  MoveL 1251 to (509.44, 499.54, 1.8) mm, rotated rx 0 ry 90 rz 0 deg; joints [-11.786, -26.31, 109.715, -15.811, -82.79, 51.021]
  Set speed (120.0 mm/s)
  MoveL 1252 to (509.32, 490.68, 1.8) mm, rotated rx 0 ry 90 rz 0 deg; joints [-10.985, -26.346, 109.945, -14.998, -82.953, 50.882]
  Set speed (30.0 mm/s)
  Call Extruder(0.767)
  MoveL 1253 to (490.68, 509.32, 1.8) mm, rotated rx 0 ry 90 rz 0 deg; joints [-13.056, -26.6, 111.69, -17.036, -84.442, 50.665]
  MoveL 1254 to (490.56, 509.44, 1.8) mm, rotated rx 0 ry 90 rz 0 deg; joints [-13.07, -26.602, 111.701, -17.049, -84.451, 50.664]
  Set speed (120.0 mm/s)
  MoveL 1255 to (490.4, 509.6, 1.8) mm, rotated rx 0 ry 90 rz 0 deg; joints [-13.088, -26.604, 111.715, -17.067, -84.463, 50.661]
  Set speed (15.0 mm/s)
  Call Extruder(0.559)
  MoveL 1256 to (490.4, 490.4, 1.8) mm, rotated rx 0 ry 90 rz 0 deg; joints [-11.303, -26.669, 112.203, -15.264, -84.829, 50.403]
  MoveL 1257 to (509.6, 490.4, 1.8) mm, rotated rx 0 ry 90 rz 0 deg; joints [-10.955, -26.341, 109.917, -14.969, -82.93, 50.884]
  MoveL 1258 to (509.6, 509.6, 1.8) mm, rotated rx 0 ry 90 rz 0 deg; joints [-12.688, -26.265, 109.434, -16.729, -82.593, 51.19]
  MoveL 1259 to (490.4, 509.6, 1.8) mm, rotated rx 0 ry 90 rz 0 deg; joints [-13.088, -26.604, 111.715, -17.067, -84.463, 50.661]
  Set speed (120.0 mm/s)
  MoveL 1260 to (490.4, 509.2, 1.8) mm, rotated rx 0 ry 90 rz 0 deg; joints [-13.051, -26.605, 111.726, -17.03, -84.471, 50.656]
  Set speed (1000.0 mm/s)
  MoveL 1261 to (491.1, 508.9, 1.8) mm, rotated rx 0 ry 90 rz 0 deg; joints [-13.008, -26.595, 111.652, -16.989, -84.409, 50.671]
  Set speed (1000.0 mm/s)
  MoveL 1262 to (490.68, 490.68, 1.8) mm, rotated rx 0 ry 90 rz 0 deg; joints [-11.324, -26.664, 112.164, -15.286, -84.797, 50.413]
  Set speed (1000.0 mm/s)
  MoveL 1263 to (490.68, 490.68, 1.9) mm, rotated rx 0 ry 90 rz 0 deg; joints [-11.324, -26.674, 112.169, -15.286, -84.792, 50.415]
  Set speed (30.0 mm/s)
  Call Extruder(0.767)
  MoveL 1264 to (509.32, 509.32, 1.9) mm, rotated rx 0 ry 90 rz 0 deg; joints [-12.669, -26.282, 109.481, -16.708, -82.621, 51.179]
  MoveL 1265 to (509.44, 509.44, 1.9) mm, rotated rx 0 ry 90 rz 0 deg; joints [-12.677, -26.279, 109.463, -16.717, -82.606, 51.185]
  Set speed (120.0 mm/s)
  MoveL 1266 to (509.32, 500.58, 1.9) mm, rotated rx 0 ry 90 rz 0 deg; joints [-11.882, -26.319, 109.709, -15.909, -82.779, 51.036]
  Set speed (30.0 mm/s)
  Call Extruder(0.360)
  MoveL 1267 to (500.58, 509.32, 1.9) mm, rotated rx 0 ry 90 rz 0 deg; joints [-12.847, -26.444, 110.525, -16.857, -83.471, 50.942]
  Set speed (120.0 mm/s)
  MoveL 1268 to (499.42, 509.32, 1.9) mm, rotated rx 0 ry 90 rz 0 deg; joints [-12.872, -26.464, 110.663, -16.877, -83.584, 50.91]
  Set speed (30.0 mm/s)
  Call Extruder(0.360)
  MoveL 1269 to (490.68, 500.58, 1.9) mm, rotated rx 0 ry 90 rz 0 deg; joints [-12.247, -26.642, 111.926, -16.218, -84.609, 50.544]
  Set speed (120.0 mm/s)
  MoveL 1270 to (490.68, 499.42, 1.9) mm, rotated rx 0 ry 90 rz 0 deg; joints [-12.139, -26.646, 111.955, -16.109, -84.631, 50.528]
  Set speed (30.0 mm/s)
  MoveL 1271 to (499.42, 490.68, 1.9) mm, rotated rx 0 ry 90 rz 0 deg; joints [-11.163, -26.533, 111.134, -15.147, -83.926, 50.637]
  Set speed (120.0 mm/s)
  MoveL 1272 to (500.58, 490.68, 1.9) mm, rotated rx 0 ry 90 rz 0 deg; joints [-11.141, -26.513, 110.996, -15.129, -83.811, 50.666]
  Set speed (30.0 mm/s)
  Call Extruder(0.360)
  MoveL 1273 to (509.32, 499.42, 1.9) mm, rotated rx 0 ry 90 rz 0 deg; joints [-11.777, -26.323, 109.738, -15.802, -82.8, 51.018]
  MoveL 1274 to (509.44, 499.54, 1.9) mm, rotated rx 0 ry 90 rz 0 deg; joints [-11.786, -26.32, 109.721, -15.812, -82.785, 51.023]
  Set speed (120.0 mm/s)
  MoveL 1275 to (509.32, 490.68, 1.9) mm, rotated rx 0 ry 90 rz 0 deg; joints [-10.985, -26.356, 109.95, -14.999, -82.948, 50.883]
  Set speed (30.0 mm/s)
  Call Extruder(0.767)
  MoveL 1276 to (490.68, 509.32, 1.9) mm, rotated rx 0 ry 90 rz 0 deg; joints [-13.056, -26.611, 111.695, -17.036, -84.437, 50.667]
  MoveL 1277 to (490.56, 509.44, 1.9) mm, rotated rx 0 ry 90 rz 0 deg; joints [-13.07, -26.612, 111.706, -17.049, -84.446, 50.665]
  Set speed (120.0 mm/s)
  MoveL 1278 to (490.4, 509.6, 1.9) mm, rotated rx 0 ry 90 rz 0 deg; joints [-13.088, -26.614, 111.72, -17.067, -84.458, 50.663]
  Set speed (15.0 mm/s)
  Call Extruder(0.559)
  MoveL 1279 to (490.4, 490.4, 1.9) mm, rotated rx 0 ry 90 rz 0 deg; joints [-11.303, -26.679, 112.209, -15.264, -84.824, 50.404]
  MoveL 1280 to (509.6, 490.4, 1.9) mm, rotated rx 0 ry 90 rz 0 deg; joints [-10.955, -26.352, 109.923, -14.969, -82.925, 50.886]
  MoveL 1281 to (509.6, 509.6, 1.9) mm, rotated rx 0 ry 90 rz 0 deg; joints [-12.688, -26.276, 109.44, -16.729, -82.588, 51.192]
  MoveL 1282 to (490.4, 509.6, 1.9) mm, rotated rx 0 ry 90 rz 0 deg; joints [-13.088, -26.614, 111.72, -17.067, -84.458, 50.663]
  Set speed (120.0 mm/s)
  MoveL 1283 to (490.4, 509.2, 1.9) mm, rotated rx 0 ry 90 rz 0 deg; joints [-13.051, -26.616, 111.731, -17.03, -84.466, 50.657]
  Set speed (1000.0 mm/s)
  MoveL 1284 to (491.1, 508.9, 1.9) mm, rotated rx 0 ry 90 rz 0 deg; joints [-13.008, -26.606, 111.657, -16.989, -84.404, 50.672]
  Set speed (1000.0 mm/s)
  MoveL 1285 to (490.68, 490.68, 1.9) mm, rotated rx 0 ry 90 rz 0 deg; joints [-11.324, -26.674, 112.169, -15.286, -84.792, 50.415]
  Set speed (1000.0 mm/s)
  MoveL 1286 to (490.68, 490.68, 2) mm, rotated rx 0 ry 90 rz 0 deg; joints [-11.324, -26.685, 112.175, -15.286, -84.786, 50.416]
  Set speed (30.0 mm/s)
  Call Extruder(0.767)
  MoveL 1287 to (509.32, 509.32, 2) mm, rotated rx 0 ry 90 rz 0 deg; joints [-12.669, -26.293, 109.486, -16.708, -82.616, 51.181]
  MoveL 1288 to (509.44, 509.44, 2) mm, rotated rx 0 ry 90 rz 0 deg; joints [-12.677, -26.29, 109.468, -16.718, -82.602, 51.186]
  Set speed (120.0 mm/s)
  MoveL 1289 to (509.32, 500.58, 2) mm, rotated rx 0 ry 90 rz 0 deg; joints [-11.882, -26.329, 109.715, -15.909, -82.774, 51.038]
  Set speed (30.0 mm/s)
  Call Extruder(0.360)
  MoveL 1290 to (500.58, 509.32, 2) mm, rotated rx 0 ry 90 rz 0 deg; joints [-12.847, -26.454, 110.53, -16.857, -83.466, 50.943]
  Set speed (120.0 mm/s)
  MoveL 1291 to (499.42, 509.32, 2) mm, rotated rx 0 ry 90 rz 0 deg; joints [-12.872, -26.475, 110.668, -16.878, -83.579, 50.911]
  Set speed (30.0 mm/s)
  Call Extruder(0.360)
  MoveL 1292 to (490.68, 500.58, 2) mm, rotated rx 0 ry 90 rz 0 deg; joints [-12.247, -26.653, 111.931, -16.218, -84.603, 50.545]
  Set speed (120.0 mm/s)
  MoveL 1293 to (490.68, 499.42, 2) mm, rotated rx 0 ry 90 rz 0 deg; joints [-12.139, -26.657, 111.961, -16.109, -84.626, 50.53]
  Set speed (30.0 mm/s)
  MoveL 1294 to (499.42, 490.68, 2) mm, rotated rx 0 ry 90 rz 0 deg; joints [-11.163, -26.543, 111.14, -15.147, -83.921, 50.638]
  Set speed (120.0 mm/s)
  MoveL 1295 to (500.58, 490.68, 2) mm, rotated rx 0 ry 90 rz 0 deg; joints [-11.141, -26.523, 111.002, -15.129, -83.806, 50.667]
  Set speed (30.0 mm/s)
  Call Extruder(0.360)
  MoveL 1296 to (509.32, 499.42, 2) mm, rotated rx 0 ry 90 rz 0 deg; joints [-11.777, -26.334, 109.744, -15.802, -82.795, 51.019]
  MoveL 1297 to (509.44, 499.54, 2) mm, rotated rx 0 ry 90 rz 0 deg; joints [-11.786, -26.331, 109.726, -15.812, -82.781, 51.024]
  Set speed (120.0 mm/s)
  MoveL 1298 to (509.32, 490.68, 2) mm, rotated rx 0 ry 90 rz 0 deg; joints [-10.985, -26.367, 109.955, -14.999, -82.943, 50.884]
  Set speed (30.0 mm/s)
  Call Extruder(0.767)
  MoveL 1299 to (490.68, 509.32, 2) mm, rotated rx 0 ry 90 rz 0 deg; joints [-13.056, -26.621, 111.7, -17.036, -84.432, 50.668]
  MoveL 1300 to (490.56, 509.44, 2) mm, rotated rx 0 ry 90 rz 0 deg; joints [-13.07, -26.623, 111.712, -17.05, -84.441, 50.667]
  Set speed (120.0 mm/s)
  MoveL 1301 to (490.4, 509.6, 2) mm, rotated rx 0 ry 90 rz 0 deg; joints [-13.088, -26.625, 111.726, -17.067, -84.453, 50.664]
  Set speed (15.0 mm/s)
  Call Extruder(0.559)
  MoveL 1302 to (490.4, 490.4, 2) mm, rotated rx 0 ry 90 rz 0 deg; joints [-11.303, -26.69, 112.214, -15.264, -84.819, 50.405]
  MoveL 1303 to (509.6, 490.4, 2) mm, rotated rx 0 ry 90 rz 0 deg; joints [-10.955, -26.362, 109.928, -14.969, -82.92, 50.887]
  MoveL 1304 to (509.6, 509.6, 2) mm, rotated rx 0 ry 90 rz 0 deg; joints [-12.688, -26.286, 109.445, -16.729, -82.583, 51.193]
  MoveL 1305 to (490.4, 509.6, 2) mm, rotated rx 0 ry 90 rz 0 deg; joints [-13.088, -26.625, 111.726, -17.067, -84.453, 50.664]
  Set speed (120.0 mm/s)
  MoveL 1306 to (490.4, 509.2, 2) mm, rotated rx 0 ry 90 rz 0 deg; joints [-13.051, -26.626, 111.737, -17.03, -84.461, 50.659]
  Set speed (1000.0 mm/s)
  MoveL 1307 to (491.1, 508.9, 2) mm, rotated rx 0 ry 90 rz 0 deg; joints [-13.008, -26.616, 111.662, -16.989, -84.399, 50.674]
  Set speed (1000.0 mm/s)
  MoveL 1308 to (490.68, 490.68, 2) mm, rotated rx 0 ry 90 rz 0 deg; joints [-11.324, -26.685, 112.175, -15.286, -84.786, 50.416]
  Set speed (1000.0 mm/s)
  MoveL 1309 to (490.68, 490.68, 2.1) mm, rotated rx 0 ry 90 rz 0 deg; joints [-11.324, -26.695, 112.18, -15.286, -84.781, 50.417]
  Set speed (30.0 mm/s)
  Call Extruder(0.767)
  MoveL 1310 to (509.32, 509.32, 2.1) mm, rotated rx 0 ry 90 rz 0 deg; joints [-12.669, -26.303, 109.491, -16.709, -82.611, 51.182]
  MoveL 1311 to (509.44, 509.44, 2.1) mm, rotated rx 0 ry 90 rz 0 deg; joints [-12.677, -26.3, 109.473, -16.718, -82.597, 51.188]
  Set speed (120.0 mm/s)
  MoveL 1312 to (509.32, 500.58, 2.1) mm, rotated rx 0 ry 90 rz 0 deg; joints [-11.882, -26.339, 109.72, -15.909, -82.769, 51.039]
  Set speed (30.0 mm/s)
  Call Extruder(0.360)
  MoveL 1313 to (500.58, 509.32, 2.1) mm, rotated rx 0 ry 90 rz 0 deg; joints [-12.847, -26.465, 110.536, -16.857, -83.462, 50.945]
  Set speed (120.0 mm/s)
  MoveL 1314 to (499.42, 509.32, 2.1) mm, rotated rx 0 ry 90 rz 0 deg; joints [-12.872, -26.485, 110.673, -16.878, -83.574, 50.913]
  Set speed (30.0 mm/s)
  Call Extruder(0.360)
  MoveL 1315 to (490.68, 500.58, 2.1) mm, rotated rx 0 ry 90 rz 0 deg; joints [-12.247, -26.663, 111.937, -16.218, -84.598, 50.547]
  Set speed (120.0 mm/s)
  MoveL 1316 to (490.68, 499.42, 2.1) mm, rotated rx 0 ry 90 rz 0 deg; joints [-12.139, -26.667, 111.966, -16.109, -84.621, 50.531]
  Set speed (30.0 mm/s)
  MoveL 1317 to (499.42, 490.68, 2.1) mm, rotated rx 0 ry 90 rz 0 deg; joints [-11.163, -26.554, 111.145, -15.147, -83.916, 50.64]
  Set speed (120.0 mm/s)
  MoveL 1318 to (500.58, 490.68, 2.1) mm, rotated rx 0 ry 90 rz 0 deg; joints [-11.141, -26.534, 111.007, -15.129, -83.801, 50.669]
  Set speed (30.0 mm/s)
  Call Extruder(0.360)
  MoveL 1319 to (509.32, 499.42, 2.1) mm, rotated rx 0 ry 90 rz 0 deg; joints [-11.777, -26.344, 109.749, -15.803, -82.79, 51.02]
  MoveL 1320 to (509.44, 499.54, 2.1) mm, rotated rx 0 ry 90 rz 0 deg; joints [-11.786, -26.341, 109.731, -15.812, -82.776, 51.026]
  Set speed (120.0 mm/s)
  MoveL 1321 to (509.32, 490.68, 2.1) mm, rotated rx 0 ry 90 rz 0 deg; joints [-10.985, -26.377, 109.961, -14.999, -82.938, 50.886]
  Set speed (30.0 mm/s)
  Call Extruder(0.767)
  MoveL 1322 to (490.68, 509.32, 2.1) mm, rotated rx 0 ry 90 rz 0 deg; joints [-13.056, -26.632, 111.706, -17.036, -84.427, 50.67]
  MoveL 1323 to (490.56, 509.44, 2.1) mm, rotated rx 0 ry 90 rz 0 deg; joints [-13.07, -26.634, 111.717, -17.05, -84.436, 50.668]
  Set speed (120.0 mm/s)
  MoveL 1324 to (490.4, 509.6, 2.1) mm, rotated rx 0 ry 90 rz 0 deg; joints [-13.088, -26.636, 111.731, -17.067, -84.448, 50.666]
  Set speed (15.0 mm/s)
  Call Extruder(0.559)
  MoveL 1325 to (490.4, 490.4, 2.1) mm, rotated rx 0 ry 90 rz 0 deg; joints [-11.303, -26.701, 112.219, -15.264, -84.814, 50.407]
  MoveL 1326 to (509.6, 490.4, 2.1) mm, rotated rx 0 ry 90 rz 0 deg; joints [-10.955, -26.373, 109.933, -14.969, -82.915, 50.888]
  MoveL 1327 to (509.6, 509.6, 2.1) mm, rotated rx 0 ry 90 rz 0 deg; joints [-12.688, -26.296, 109.45, -16.729, -82.578, 51.195]
  MoveL 1328 to (490.4, 509.6, 2.1) mm, rotated rx 0 ry 90 rz 0 deg; joints [-13.088, -26.636, 111.731, -17.067, -84.448, 50.666]
  Set speed (120.0 mm/s)
  MoveL 1329 to (490.4, 509.2, 2.1) mm, rotated rx 0 ry 90 rz 0 deg; joints [-13.051, -26.637, 111.742, -17.03, -84.456, 50.66]
  Set speed (1000.0 mm/s)
  MoveL 1330 to (491.1, 508.9, 2.1) mm, rotated rx 0 ry 90 rz 0 deg; joints [-13.008, -26.627, 111.668, -16.989, -84.394, 50.676]
  Set speed (1000.0 mm/s)
  MoveL 1331 to (490.68, 490.68, 2.1) mm, rotated rx 0 ry 90 rz 0 deg; joints [-11.324, -26.695, 112.18, -15.286, -84.781, 50.417]
  Set speed (1000.0 mm/s)
  MoveL 1332 to (490.68, 490.68, 2.2) mm, rotated rx 0 ry 90 rz 0 deg; joints [-11.324, -26.706, 112.185, -15.286, -84.776, 50.419]
  Set speed (30.0 mm/s)
  Call Extruder(0.767)
  MoveL 1333 to (509.32, 509.32, 2.2) mm, rotated rx 0 ry 90 rz 0 deg; joints [-12.669, -26.314, 109.497, -16.709, -82.606, 51.184]
  MoveL 1334 to (509.44, 509.44, 2.2) mm, rotated rx 0 ry 90 rz 0 deg; joints [-12.677, -26.311, 109.479, -16.718, -82.592, 51.189]
  Set speed (120.0 mm/s)
  MoveL 1335 to (509.32, 500.58, 2.2) mm, rotated rx 0 ry 90 rz 0 deg; joints [-11.882, -26.35, 109.725, -15.909, -82.765, 51.04]
  Set speed (30.0 mm/s)
  Call Extruder(0.360)
  MoveL 1336 to (500.58, 509.32, 2.2) mm, rotated rx 0 ry 90 rz 0 deg; joints [-12.847, -26.475, 110.541, -16.858, -83.457, 50.946]
  Set speed (120.0 mm/s)
  MoveL 1337 to (499.42, 509.32, 2.2) mm, rotated rx 0 ry 90 rz 0 deg; joints [-12.872, -26.496, 110.679, -16.878, -83.569, 50.914]
  Set speed (30.0 mm/s)
  Call Extruder(0.360)
  MoveL 1338 to (490.68, 500.58, 2.2) mm, rotated rx 0 ry 90 rz 0 deg; joints [-12.247, -26.674, 111.942, -16.218, -84.593, 50.548]
  Set speed (120.0 mm/s)
  MoveL 1339 to (490.68, 499.42, 2.2) mm, rotated rx 0 ry 90 rz 0 deg; joints [-12.139, -26.678, 111.972, -16.109, -84.616, 50.533]
  Set speed (30.0 mm/s)
  MoveL 1340 to (499.42, 490.68, 2.2) mm, rotated rx 0 ry 90 rz 0 deg; joints [-11.163, -26.564, 111.15, -15.147, -83.911, 50.641]
  Set speed (120.0 mm/s)
  MoveL 1341 to (500.58, 490.68, 2.2) mm, rotated rx 0 ry 90 rz 0 deg; joints [-11.141, -26.545, 111.012, -15.129, -83.796, 50.67]
  Set speed (30.0 mm/s)
  Call Extruder(0.360)
  MoveL 1342 to (509.32, 499.42, 2.2) mm, rotated rx 0 ry 90 rz 0 deg; joints [-11.777, -26.355, 109.754, -15.803, -82.785, 51.022]
  MoveL 1343 to (509.44, 499.54, 2.2) mm, rotated rx 0 ry 90 rz 0 deg; joints [-11.786, -26.352, 109.737, -15.812, -82.771, 51.027]
  Set speed (120.0 mm/s)
  MoveL 1344 to (509.32, 490.68, 2.2) mm, rotated rx 0 ry 90 rz 0 deg; joints [-10.985, -26.388, 109.966, -14.999, -82.933, 50.887]
  Set speed (30.0 mm/s)
  Call Extruder(0.767)
  MoveL 1345 to (490.68, 509.32, 2.2) mm, rotated rx 0 ry 90 rz 0 deg; joints [-13.056, -26.643, 111.711, -17.036, -84.422, 50.671]
  MoveL 1346 to (490.56, 509.44, 2.2) mm, rotated rx 0 ry 90 rz 0 deg; joints [-13.07, -26.644, 111.722, -17.05, -84.431, 50.67]
  Set speed (120.0 mm/s)
  MoveL 1347 to (490.4, 509.6, 2.2) mm, rotated rx 0 ry 90 rz 0 deg; joints [-13.088, -26.646, 111.736, -17.068, -84.443, 50.668]
  Set speed (15.0 mm/s)
  Call Extruder(0.559)
  MoveL 1348 to (490.4, 490.4, 2.2) mm, rotated rx 0 ry 90 rz 0 deg; joints [-11.303, -26.711, 112.225, -15.264, -84.809, 50.408]
  MoveL 1349 to (509.6, 490.4, 2.2) mm, rotated rx 0 ry 90 rz 0 deg; joints [-10.955, -26.383, 109.939, -14.969, -82.91, 50.89]
  MoveL 1350 to (509.6, 509.6, 2.2) mm, rotated rx 0 ry 90 rz 0 deg; joints [-12.688, -26.307, 109.456, -16.73, -82.574, 51.196]
  MoveL 1351 to (490.4, 509.6, 2.2) mm, rotated rx 0 ry 90 rz 0 deg; joints [-13.088, -26.646, 111.736, -17.068, -84.443, 50.668]
  Set speed (120.0 mm/s)
  MoveL 1352 to (490.4, 509.2, 2.2) mm, rotated rx 0 ry 90 rz 0 deg; joints [-13.051, -26.648, 111.747, -17.03, -84.451, 50.662]
  Set speed (1000.0 mm/s)
  MoveL 1353 to (491.1, 508.9, 2.2) mm, rotated rx 0 ry 90 rz 0 deg; joints [-13.008, -26.637, 111.673, -16.989, -84.389, 50.677]
  Set speed (1000.0 mm/s)
  MoveL 1354 to (490.68, 490.68, 2.2) mm, rotated rx 0 ry 90 rz 0 deg; joints [-11.324, -26.706, 112.185, -15.286, -84.776, 50.419]
  Set speed (1000.0 mm/s)
  MoveL 1355 to (490.68, 490.68, 2.3) mm, rotated rx 0 ry 90 rz 0 deg; joints [-11.324, -26.717, 112.191, -15.286, -84.771, 50.42]
  Set speed (30.0 mm/s)
  Call Extruder(0.767)
  MoveL 1356 to (509.32, 509.32, 2.3) mm, rotated rx 0 ry 90 rz 0 deg; joints [-12.669, -26.324, 109.502, -16.709, -82.601, 51.185]
  MoveL 1357 to (509.44, 509.44, 2.3) mm, rotated rx 0 ry 90 rz 0 deg; joints [-12.677, -26.321, 109.484, -16.718, -82.587, 51.191]
  Set speed (120.0 mm/s)
  MoveL 1358 to (509.32, 500.58, 2.3) mm, rotated rx 0 ry 90 rz 0 deg; joints [-11.882, -26.36, 109.731, -15.909, -82.76, 51.042]
  Set speed (30.0 mm/s)
  Call Extruder(0.360)
  MoveL 1359 to (500.58, 509.32, 2.3) mm, rotated rx 0 ry 90 rz 0 deg; joints [-12.847, -26.486, 110.546, -16.858, -83.452, 50.948]
  Set speed (120.0 mm/s)
  MoveL 1360 to (499.42, 509.32, 2.3) mm, rotated rx 0 ry 90 rz 0 deg; joints [-12.872, -26.506, 110.684, -16.878, -83.565, 50.916]
  Set speed (30.0 mm/s)
  Call Extruder(0.360)
  MoveL 1361 to (490.68, 500.58, 2.3) mm, rotated rx 0 ry 90 rz 0 deg; joints [-12.247, -26.685, 111.947, -16.218, -84.588, 50.55]
  Set speed (120.0 mm/s)
  MoveL 1362 to (490.68, 499.42, 2.3) mm, rotated rx 0 ry 90 rz 0 deg; joints [-12.139, -26.688, 111.977, -16.109, -84.61, 50.534]
  Set speed (30.0 mm/s)
  MoveL 1363 to (499.42, 490.68, 2.3) mm, rotated rx 0 ry 90 rz 0 deg; joints [-11.163, -26.575, 111.156, -15.147, -83.906, 50.642]
  Set speed (120.0 mm/s)
  MoveL 1364 to (500.58, 490.68, 2.3) mm, rotated rx 0 ry 90 rz 0 deg; joints [-11.141, -26.555, 111.018, -15.13, -83.791, 50.671]
  Set speed (30.0 mm/s)
  Call Extruder(0.360)
  MoveL 1365 to (509.32, 499.42, 2.3) mm, rotated rx 0 ry 90 rz 0 deg; joints [-11.777, -26.365, 109.76, -15.803, -82.78, 51.023]
  MoveL 1366 to (509.44, 499.54, 2.3) mm, rotated rx 0 ry 90 rz 0 deg; joints [-11.786, -26.362, 109.742, -15.812, -82.766, 51.028]
  Set speed (120.0 mm/s)
  MoveL 1367 to (509.32, 490.68, 2.3) mm, rotated rx 0 ry 90 rz 0 deg; joints [-10.985, -26.398, 109.971, -14.999, -82.928, 50.888]
  Set speed (30.0 mm/s)
  Call Extruder(0.767)
  MoveL 1368 to (490.68, 509.32, 2.3) mm, rotated rx 0 ry 90 rz 0 deg; joints [-13.056, -26.653, 111.717, -17.036, -84.417, 50.673]
  MoveL 1369 to (490.56, 509.44, 2.3) mm, rotated rx 0 ry 90 rz 0 deg; joints [-13.07, -26.655, 111.728, -17.05, -84.426, 50.671]
  Set speed (120.0 mm/s)
  MoveL 1370 to (490.4, 509.6, 2.3) mm, rotated rx 0 ry 90 rz 0 deg; joints [-13.088, -26.657, 111.742, -17.068, -84.438, 50.669]
  Set speed (15.0 mm/s)
  Call Extruder(0.559)
  MoveL 1371 to (490.4, 490.4, 2.3) mm, rotated rx 0 ry 90 rz 0 deg; joints [-11.303, -26.722, 112.23, -15.265, -84.804, 50.41]
  MoveL 1372 to (509.6, 490.4, 2.3) mm, rotated rx 0 ry 90 rz 0 deg; joints [-10.955, -26.394, 109.944, -14.969, -82.905, 50.891]
  MoveL 1373 to (509.6, 509.6, 2.3) mm, rotated rx 0 ry 90 rz 0 deg; joints [-12.688, -26.317, 109.461, -16.73, -82.569, 51.198]
  MoveL 1374 to (490.4, 509.6, 2.3) mm, rotated rx 0 ry 90 rz 0 deg; joints [-13.088, -26.657, 111.742, -17.068, -84.438, 50.669]
  Set speed (120.0 mm/s)
  MoveL 1375 to (490.4, 509.2, 2.3) mm, rotated rx 0 ry 90 rz 0 deg; joints [-13.051, -26.658, 111.753, -17.03, -84.446, 50.663]
  Set speed (1000.0 mm/s)
  MoveL 1376 to (491.1, 508.9, 2.3) mm, rotated rx 0 ry 90 rz 0 deg; joints [-13.008, -26.648, 111.679, -16.989, -84.384, 50.679]
  Set speed (1000.0 mm/s)
  MoveL 1377 to (490.68, 490.68, 2.3) mm, rotated rx 0 ry 90 rz 0 deg; joints [-11.324, -26.717, 112.191, -15.286, -84.771, 50.42]
  Set speed (1000.0 mm/s)
  MoveL 1378 to (490.68, 490.68, 2.4) mm, rotated rx 0 ry 90 rz 0 deg; joints [-11.324, -26.727, 112.196, -15.286, -84.766, 50.422]
  Set speed (30.0 mm/s)
  Call Extruder(0.767)
  MoveL 1379 to (509.32, 509.32, 2.4) mm, rotated rx 0 ry 90 rz 0 deg; joints [-12.669, -26.334, 109.507, -16.709, -82.596, 51.187]
  MoveL 1380 to (509.44, 509.44, 2.4) mm, rotated rx 0 ry 90 rz 0 deg; joints [-12.677, -26.332, 109.489, -16.718, -82.582, 51.192]
  Set speed (120.0 mm/s)
  MoveL 1381 to (509.32, 500.58, 2.4) mm, rotated rx 0 ry 90 rz 0 deg; joints [-11.882, -26.371, 109.736, -15.909, -82.755, 51.043]
  Set speed (30.0 mm/s)
  Call Extruder(0.360)
  MoveL 1382 to (500.58, 509.32, 2.4) mm, rotated rx 0 ry 90 rz 0 deg; joints [-12.847, -26.496, 110.552, -16.858, -83.447, 50.949]
  Set speed (120.0 mm/s)
  MoveL 1383 to (499.42, 509.32, 2.4) mm, rotated rx 0 ry 90 rz 0 deg; joints [-12.872, -26.517, 110.689, -16.878, -83.56, 50.917]
  Set speed (30.0 mm/s)
  Call Extruder(0.360)
  MoveL 1384 to (490.68, 500.58, 2.4) mm, rotated rx 0 ry 90 rz 0 deg; joints [-12.247, -26.695, 111.953, -16.218, -84.583, 50.551]
  Set speed (120.0 mm/s)
  MoveL 1385 to (490.68, 499.42, 2.4) mm, rotated rx 0 ry 90 rz 0 deg; joints [-12.139, -26.699, 111.982, -16.109, -84.605, 50.536]
  Set speed (30.0 mm/s)
  MoveL 1386 to (499.42, 490.68, 2.4) mm, rotated rx 0 ry 90 rz 0 deg; joints [-11.163, -26.586, 111.161, -15.148, -83.901, 50.644]
  Set speed (120.0 mm/s)
  MoveL 1387 to (500.58, 490.68, 2.4) mm, rotated rx 0 ry 90 rz 0 deg; joints [-11.141, -26.566, 111.023, -15.13, -83.786, 50.673]
  Set speed (30.0 mm/s)
  Call Extruder(0.360)
  MoveL 1388 to (509.32, 499.42, 2.4) mm, rotated rx 0 ry 90 rz 0 deg; joints [-11.777, -26.375, 109.765, -15.803, -82.775, 51.025]
  MoveL 1389 to (509.44, 499.54, 2.4) mm, rotated rx 0 ry 90 rz 0 deg; joints [-11.786, -26.373, 109.747, -15.812, -82.761, 51.03]
  Set speed (120.0 mm/s)
  MoveL 1390 to (509.32, 490.68, 2.4) mm, rotated rx 0 ry 90 rz 0 deg; joints [-10.985, -26.409, 109.977, -14.999, -82.923, 50.89]
  Set speed (30.0 mm/s)
  Call Extruder(0.767)
  MoveL 1391 to (490.68, 509.32, 2.4) mm, rotated rx 0 ry 90 rz 0 deg; joints [-13.056, -26.664, 111.722, -17.036, -84.412, 50.674]
  MoveL 1392 to (490.56, 509.44, 2.4) mm, rotated rx 0 ry 90 rz 0 deg; joints [-13.07, -26.665, 111.733, -17.05, -84.421, 50.673]
  Set speed (120.0 mm/s)
  MoveL 1393 to (490.4, 509.6, 2.4) mm, rotated rx 0 ry 90 rz 0 deg; joints [-13.088, -26.667, 111.747, -17.068, -84.433, 50.671]
  Set speed (15.0 mm/s)
  Call Extruder(0.559)
  MoveL 1394 to (490.4, 490.4, 2.4) mm, rotated rx 0 ry 90 rz 0 deg; joints [-11.303, -26.733, 112.236, -15.265, -84.799, 50.411]
  MoveL 1395 to (509.6, 490.4, 2.4) mm, rotated rx 0 ry 90 rz 0 deg; joints [-10.955, -26.404, 109.949, -14.97, -82.9, 50.892]
  MoveL 1396 to (509.6, 509.6, 2.4) mm, rotated rx 0 ry 90 rz 0 deg; joints [-12.688, -26.328, 109.466, -16.73, -82.564, 51.199]
  MoveL 1397 to (490.4, 509.6, 2.4) mm, rotated rx 0 ry 90 rz 0 deg; joints [-13.088, -26.667, 111.747, -17.068, -84.433, 50.671]
  Set speed (120.0 mm/s)
  MoveL 1398 to (490.4, 509.2, 2.4) mm, rotated rx 0 ry 90 rz 0 deg; joints [-13.051, -26.669, 111.758, -17.031, -84.441, 50.665]
  Set speed (1000.0 mm/s)
  MoveL 1399 to (491.1, 508.9, 2.4) mm, rotated rx 0 ry 90 rz 0 deg; joints [-13.008, -26.659, 111.684, -16.99, -84.379, 50.68]
  Set speed (1000.0 mm/s)
  MoveL 1400 to (490.68, 490.68, 2.4) mm, rotated rx 0 ry 90 rz 0 deg; joints [-11.324, -26.727, 112.196, -15.286, -84.766, 50.422]
  Set speed (1000.0 mm/s)
  MoveL 1401 to (490.68, 490.68, 2.5) mm, rotated rx 0 ry 90 rz 0 deg; joints [-11.324, -26.738, 112.202, -15.287, -84.761, 50.423]
  Set speed (30.0 mm/s)
  Call Extruder(0.767)
  MoveL 1402 to (509.32, 509.32, 2.5) mm, rotated rx 0 ry 90 rz 0 deg; joints [-12.669, -26.345, 109.513, -16.709, -82.591, 51.188]
  MoveL 1403 to (509.44, 509.44, 2.5) mm, rotated rx 0 ry 90 rz 0 deg; joints [-12.677, -26.342, 109.495, -16.718, -82.577, 51.194]
  Set speed (120.0 mm/s)
  MoveL 1404 to (509.32, 500.58, 2.5) mm, rotated rx 0 ry 90 rz 0 deg; joints [-11.882, -26.381, 109.741, -15.91, -82.75, 51.045]
  Set speed (30.0 mm/s)
  Call Extruder(0.360)
  MoveL 1405 to (500.58, 509.32, 2.5) mm, rotated rx 0 ry 90 rz 0 deg; joints [-12.847, -26.507, 110.557, -16.858, -83.442, 50.951]
  Set speed (120.0 mm/s)
  MoveL 1406 to (499.42, 509.32, 2.5) mm, rotated rx 0 ry 90 rz 0 deg; joints [-12.872, -26.527, 110.695, -16.878, -83.555, 50.919]
  Set speed (30.0 mm/s)
  Call Extruder(0.360)
  MoveL 1407 to (490.68, 500.58, 2.5) mm, rotated rx 0 ry 90 rz 0 deg; joints [-12.247, -26.706, 111.958, -16.218, -84.578, 50.553]
  Set speed (120.0 mm/s)
  MoveL 1408 to (490.68, 499.42, 2.5) mm, rotated rx 0 ry 90 rz 0 deg; joints [-12.139, -26.71, 111.988, -16.109, -84.6, 50.537]
  Set speed (30.0 mm/s)
  MoveL 1409 to (499.42, 490.68, 2.5) mm, rotated rx 0 ry 90 rz 0 deg; joints [-11.163, -26.596, 111.166, -15.148, -83.896, 50.645]
  Set speed (120.0 mm/s)
  MoveL 1410 to (500.58, 490.68, 2.5) mm, rotated rx 0 ry 90 rz 0 deg; joints [-11.141, -26.576, 111.028, -15.13, -83.781, 50.674]
  Set speed (30.0 mm/s)
  Call Extruder(0.360)
  MoveL 1411 to (509.32, 499.42, 2.5) mm, rotated rx 0 ry 90 rz 0 deg; joints [-11.777, -26.386, 109.77, -15.803, -82.77, 51.026]
  MoveL 1412 to (509.44, 499.54, 2.5) mm, rotated rx 0 ry 90 rz 0 deg; joints [-11.786, -26.383, 109.753, -15.813, -82.756, 51.031]
  Set speed (120.0 mm/s)
  MoveL 1413 to (509.32, 490.68, 2.5) mm, rotated rx 0 ry 90 rz 0 deg; joints [-10.985, -26.419, 109.982, -15, -82.918, 50.891]
  Set speed (30.0 mm/s)
  Call Extruder(0.767)
  MoveL 1414 to (490.68, 509.32, 2.5) mm, rotated rx 0 ry 90 rz 0 deg; joints [-13.056, -26.675, 111.727, -17.037, -84.407, 50.676]
  MoveL 1415 to (490.56, 509.44, 2.5) mm, rotated rx 0 ry 90 rz 0 deg; joints [-13.07, -26.676, 111.739, -17.05, -84.416, 50.674]
  Set speed (120.0 mm/s)
  MoveL 1416 to (490.4, 509.6, 2.5) mm, rotated rx 0 ry 90 rz 0 deg; joints [-13.088, -26.678, 111.753, -17.068, -84.428, 50.672]
  Set speed (15.0 mm/s)
  Call Extruder(0.559)
  MoveL 1417 to (490.4, 490.4, 2.5) mm, rotated rx 0 ry 90 rz 0 deg; joints [-11.303, -26.743, 112.241, -15.265, -84.794, 50.412]
  MoveL 1418 to (509.6, 490.4, 2.5) mm, rotated rx 0 ry 90 rz 0 deg; joints [-10.955, -26.415, 109.955, -14.97, -82.895, 50.894]
  MoveL 1419 to (509.6, 509.6, 2.5) mm, rotated rx 0 ry 90 rz 0 deg; joints [-12.688, -26.338, 109.471, -16.73, -82.559, 51.201]
  MoveL 1420 to (490.4, 509.6, 2.5) mm, rotated rx 0 ry 90 rz 0 deg; joints [-13.088, -26.678, 111.753, -17.068, -84.428, 50.672]
  Set speed (120.0 mm/s)
  MoveL 1421 to (490.4, 509.2, 2.5) mm, rotated rx 0 ry 90 rz 0 deg; joints [-13.051, -26.679, 111.763, -17.031, -84.436, 50.666]
  Set speed (1000.0 mm/s)
  MoveL 1422 to (491.1, 508.9, 2.5) mm, rotated rx 0 ry 90 rz 0 deg; joints [-13.008, -26.669, 111.689, -16.99, -84.374, 50.682]
  Set speed (1000.0 mm/s)
  MoveL 1423 to (490.68, 490.68, 2.5) mm, rotated rx 0 ry 90 rz 0 deg; joints [-11.324, -26.738, 112.202, -15.287, -84.761, 50.423]
  Set speed (1000.0 mm/s)
  MoveL 1424 to (490.68, 490.68, 2.6) mm, rotated rx 0 ry 90 rz 0 deg; joints [-11.324, -26.749, 112.207, -15.287, -84.756, 50.424]
  Set speed (30.0 mm/s)
  Call Extruder(0.767)
  MoveL 1425 to (509.32, 509.32, 2.6) mm, rotated rx 0 ry 90 rz 0 deg; joints [-12.669, -26.355, 109.518, -16.709, -82.586, 51.19]
  MoveL 1426 to (509.44, 509.44, 2.6) mm, rotated rx 0 ry 90 rz 0 deg; joints [-12.677, -26.352, 109.5, -16.719, -82.572, 51.195]
  Set speed (120.0 mm/s)
  MoveL 1427 to (509.32, 500.58, 2.6) mm, rotated rx 0 ry 90 rz 0 deg; joints [-11.882, -26.392, 109.747, -15.91, -82.745, 51.046]
  Set speed (30.0 mm/s)
  Call Extruder(0.360)
  MoveL 1428 to (500.58, 509.32, 2.6) mm, rotated rx 0 ry 90 rz 0 deg; joints [-12.847, -26.517, 110.562, -16.858, -83.437, 50.952]
  Set speed (120.0 mm/s)
  MoveL 1429 to (499.42, 509.32, 2.6) mm, rotated rx 0 ry 90 rz 0 deg; joints [-12.872, -26.538, 110.7, -16.879, -83.55, 50.92]
  Set speed (30.0 mm/s)
  Call Extruder(0.360)
  MoveL 1430 to (490.68, 500.58, 2.6) mm, rotated rx 0 ry 90 rz 0 deg; joints [-12.247, -26.716, 111.964, -16.218, -84.573, 50.554]
  Set speed (120.0 mm/s)
  MoveL 1431 to (490.68, 499.42, 2.6) mm, rotated rx 0 ry 90 rz 0 deg; joints [-12.139, -26.72, 111.993, -16.11, -84.595, 50.538]
  Set speed (30.0 mm/s)
  MoveL 1432 to (499.42, 490.68, 2.6) mm, rotated rx 0 ry 90 rz 0 deg; joints [-11.163, -26.607, 111.172, -15.148, -83.891, 50.646]
  Set speed (120.0 mm/s)
  MoveL 1433 to (500.58, 490.68, 2.6) mm, rotated rx 0 ry 90 rz 0 deg; joints [-11.141, -26.587, 111.034, -15.13, -83.776, 50.675]
  Set speed (30.0 mm/s)
  Call Extruder(0.360)
  MoveL 1434 to (509.32, 499.42, 2.6) mm, rotated rx 0 ry 90 rz 0 deg; joints [-11.777, -26.396, 109.776, -15.803, -82.765, 51.028]
  MoveL 1435 to (509.44, 499.54, 2.6) mm, rotated rx 0 ry 90 rz 0 deg; joints [-11.786, -26.394, 109.758, -15.813, -82.751, 51.033]
  Set speed (120.0 mm/s)
  MoveL 1436 to (509.32, 490.68, 2.6) mm, rotated rx 0 ry 90 rz 0 deg; joints [-10.985, -26.43, 109.987, -15, -82.913, 50.892]
  Set speed (30.0 mm/s)
  Call Extruder(0.767)
  MoveL 1437 to (490.68, 509.32, 2.6) mm, rotated rx 0 ry 90 rz 0 deg; joints [-13.056, -26.685, 111.733, -17.037, -84.402, 50.677]
  MoveL 1438 to (490.56, 509.44, 2.6) mm, rotated rx 0 ry 90 rz 0 deg; joints [-13.07, -26.687, 111.744, -17.051, -84.411, 50.676]
  Set speed (120.0 mm/s)
  MoveL 1439 to (490.4, 509.6, 2.6) mm, rotated rx 0 ry 90 rz 0 deg; joints [-13.088, -26.689, 111.758, -17.068, -84.423, 50.674]
  Set speed (15.0 mm/s)
  Call Extruder(0.559)
  MoveL 1440 to (490.4, 490.4, 2.6) mm, rotated rx 0 ry 90 rz 0 deg; joints [-11.303, -26.754, 112.246, -15.265, -84.789, 50.414]
  MoveL 1441 to (509.6, 490.4, 2.6) mm, rotated rx 0 ry 90 rz 0 deg; joints [-10.955, -26.425, 109.96, -14.97, -82.89, 50.895]
  MoveL 1442 to (509.6, 509.6, 2.6) mm, rotated rx 0 ry 90 rz 0 deg; joints [-12.688, -26.349, 109.477, -16.73, -82.554, 51.202]
  MoveL 1443 to (490.4, 509.6, 2.6) mm, rotated rx 0 ry 90 rz 0 deg; joints [-13.088, -26.689, 111.758, -17.068, -84.423, 50.674]
  Set speed (120.0 mm/s)
  MoveL 1444 to (490.4, 509.2, 2.6) mm, rotated rx 0 ry 90 rz 0 deg; joints [-13.051, -26.69, 111.769, -17.031, -84.431, 50.668]
  Set speed (1000.0 mm/s)
  MoveL 1445 to (491.1, 508.9, 2.6) mm, rotated rx 0 ry 90 rz 0 deg; joints [-13.008, -26.68, 111.695, -16.99, -84.369, 50.683]
  Set speed (1000.0 mm/s)
  MoveL 1446 to (490.68, 490.68, 2.6) mm, rotated rx 0 ry 90 rz 0 deg; joints [-11.324, -26.749, 112.207, -15.287, -84.756, 50.424]
  Set speed (1000.0 mm/s)
  MoveL 1447 to (490.68, 490.68, 2.7) mm, rotated rx 0 ry 90 rz 0 deg; joints [-11.324, -26.759, 112.212, -15.287, -84.751, 50.426]
  Set speed (30.0 mm/s)
  Call Extruder(0.767)
  MoveL 1448 to (509.32, 509.32, 2.7) mm, rotated rx 0 ry 90 rz 0 deg; joints [-12.669, -26.366, 109.523, -16.71, -82.582, 51.191]
  MoveL 1449 to (509.44, 509.44, 2.7) mm, rotated rx 0 ry 90 rz 0 deg; joints [-12.677, -26.363, 109.505, -16.719, -82.567, 51.197]
  Set speed (120.0 mm/s)
  MoveL 1450 to (509.32, 500.58, 2.7) mm, rotated rx 0 ry 90 rz 0 deg; joints [-11.882, -26.402, 109.752, -15.91, -82.74, 51.047]
  Set speed (30.0 mm/s)
  Call Extruder(0.360)
  MoveL 1451 to (500.58, 509.32, 2.7) mm, rotated rx 0 ry 90 rz 0 deg; joints [-12.847, -26.528, 110.568, -16.858, -83.432, 50.954]
  Set speed (120.0 mm/s)
  MoveL 1452 to (499.42, 509.32, 2.7) mm, rotated rx 0 ry 90 rz 0 deg; joints [-12.872, -26.548, 110.705, -16.879, -83.545, 50.922]
  Set speed (30.0 mm/s)
  Call Extruder(0.360)
  MoveL 1453 to (490.68, 500.58, 2.7) mm, rotated rx 0 ry 90 rz 0 deg; joints [-12.247, -26.727, 111.969, -16.219, -84.568, 50.556]
  Set speed (120.0 mm/s)
  MoveL 1454 to (490.68, 499.42, 2.7) mm, rotated rx 0 ry 90 rz 0 deg; joints [-12.139, -26.731, 111.999, -16.11, -84.59, 50.54]
  Set speed (30.0 mm/s)
  MoveL 1455 to (499.42, 490.68, 2.7) mm, rotated rx 0 ry 90 rz 0 deg; joints [-11.163, -26.617, 111.177, -15.148, -83.886, 50.648]
  Set speed (120.0 mm/s)
  MoveL 1456 to (500.58, 490.68, 2.7) mm, rotated rx 0 ry 90 rz 0 deg; joints [-11.141, -26.597, 111.039, -15.13, -83.771, 50.677]
  Set speed (30.0 mm/s)
  Call Extruder(0.360)
  MoveL 1457 to (509.32, 499.42, 2.7) mm, rotated rx 0 ry 90 rz 0 deg; joints [-11.777, -26.407, 109.781, -15.804, -82.76, 51.029]
  MoveL 1458 to (509.44, 499.54, 2.7) mm, rotated rx 0 ry 90 rz 0 deg; joints [-11.786, -26.404, 109.763, -15.813, -82.746, 51.034]
  Set speed (120.0 mm/s)
  MoveL 1459 to (509.32, 490.68, 2.7) mm, rotated rx 0 ry 90 rz 0 deg; joints [-10.985, -26.44, 109.993, -15, -82.908, 50.894]
  Set speed (30.0 mm/s)
  Call Extruder(0.767)
  MoveL 1460 to (490.68, 509.32, 2.7) mm, rotated rx 0 ry 90 rz 0 deg; joints [-13.056, -26.696, 111.738, -17.037, -84.397, 50.679]
  MoveL 1461 to (490.56, 509.44, 2.7) mm, rotated rx 0 ry 90 rz 0 deg; joints [-13.07, -26.697, 111.749, -17.051, -84.406, 50.677]
  Set speed (120.0 mm/s)
  MoveL 1462 to (490.4, 509.6, 2.7) mm, rotated rx 0 ry 90 rz 0 deg; joints [-13.088, -26.699, 111.763, -17.068, -84.418, 50.675]
  Set speed (15.0 mm/s)
  Call Extruder(0.559)
  MoveL 1463 to (490.4, 490.4, 2.7) mm, rotated rx 0 ry 90 rz 0 deg; joints [-11.303, -26.765, 112.252, -15.265, -84.784, 50.415]
  MoveL 1464 to (509.6, 490.4, 2.7) mm, rotated rx 0 ry 90 rz 0 deg; joints [-10.955, -26.436, 109.965, -14.97, -82.885, 50.896]
  MoveL 1465 to (509.6, 509.6, 2.7) mm, rotated rx 0 ry 90 rz 0 deg; joints [-12.688, -26.359, 109.482, -16.731, -82.549, 51.204]
  MoveL 1466 to (490.4, 509.6, 2.7) mm, rotated rx 0 ry 90 rz 0 deg; joints [-13.088, -26.699, 111.763, -17.068, -84.418, 50.675]
  Set speed (120.0 mm/s)
  MoveL 1467 to (490.4, 509.2, 2.7) mm, rotated rx 0 ry 90 rz 0 deg; joints [-13.051, -26.701, 111.774, -17.031, -84.426, 50.669]
  Set speed (1000.0 mm/s)
  MoveL 1468 to (491.1, 508.9, 2.7) mm, rotated rx 0 ry 90 rz 0 deg; joints [-13.008, -26.691, 111.7, -16.99, -84.364, 50.685]
  Set speed (1000.0 mm/s)
  MoveL 1469 to (490.68, 490.68, 2.7) mm, rotated rx 0 ry 90 rz 0 deg; joints [-11.324, -26.759, 112.212, -15.287, -84.751, 50.426]
  Set speed (1000.0 mm/s)
  MoveL 1470 to (490.68, 490.68, 2.8) mm, rotated rx 0 ry 90 rz 0 deg; joints [-11.324, -26.77, 112.218, -15.287, -84.746, 50.427]
  Set speed (30.0 mm/s)
  Call Extruder(0.767)
  MoveL 1471 to (509.32, 509.32, 2.8) mm, rotated rx 0 ry 90 rz 0 deg; joints [-12.669, -26.376, 109.529, -16.71, -82.577, 51.193]
  MoveL 1472 to (509.44, 509.44, 2.8) mm, rotated rx 0 ry 90 rz 0 deg; joints [-12.677, -26.373, 109.511, -16.719, -82.562, 51.198]
  Set speed (120.0 mm/s)
  MoveL 1473 to (509.32, 500.58, 2.8) mm, rotated rx 0 ry 90 rz 0 deg; joints [-11.882, -26.413, 109.757, -15.91, -82.735, 51.049]
  Set speed (30.0 mm/s)
  Call Extruder(0.360)
  MoveL 1474 to (500.58, 509.32, 2.8) mm, rotated rx 0 ry 90 rz 0 deg; joints [-12.847, -26.538, 110.573, -16.859, -83.427, 50.955]
  Set speed (120.0 mm/s)
  MoveL 1475 to (499.42, 509.32, 2.8) mm, rotated rx 0 ry 90 rz 0 deg; joints [-12.872, -26.559, 110.711, -16.879, -83.54, 50.924]
  Set speed (30.0 mm/s)
  Call Extruder(0.360)
  MoveL 1476 to (490.68, 500.58, 2.8) mm, rotated rx 0 ry 90 rz 0 deg; joints [-12.247, -26.738, 111.974, -16.219, -84.563, 50.557]
  Set speed (120.0 mm/s)
  MoveL 1477 to (490.68, 499.42, 2.8) mm, rotated rx 0 ry 90 rz 0 deg; joints [-12.139, -26.742, 112.004, -16.11, -84.585, 50.541]
  Set speed (30.0 mm/s)
  MoveL 1478 to (499.42, 490.68, 2.8) mm, rotated rx 0 ry 90 rz 0 deg; joints [-11.163, -26.628, 111.183, -15.148, -83.881, 50.649]
  Set speed (120.0 mm/s)
  MoveL 1479 to (500.58, 490.68, 2.8) mm, rotated rx 0 ry 90 rz 0 deg; joints [-11.141, -26.608, 111.044, -15.13, -83.766, 50.678]
  Set speed (30.0 mm/s)
  Call Extruder(0.360)
  MoveL 1480 to (509.32, 499.42, 2.8) mm, rotated rx 0 ry 90 rz 0 deg; joints [-11.777, -26.417, 109.786, -15.804, -82.755, 51.03]
  MoveL 1481 to (509.44, 499.54, 2.8) mm, rotated rx 0 ry 90 rz 0 deg; joints [-11.786, -26.414, 109.769, -15.813, -82.741, 51.035]
  Set speed (120.0 mm/s)
  MoveL 1482 to (509.32, 490.68, 2.8) mm, rotated rx 0 ry 90 rz 0 deg; joints [-10.985, -26.45, 109.998, -15, -82.903, 50.895]
  Set speed (30.0 mm/s)
  Call Extruder(0.767)
  MoveL 1483 to (490.68, 509.32, 2.8) mm, rotated rx 0 ry 90 rz 0 deg; joints [-13.056, -26.706, 111.744, -17.037, -84.392, 50.681]
  MoveL 1484 to (490.56, 509.44, 2.8) mm, rotated rx 0 ry 90 rz 0 deg; joints [-13.07, -26.708, 111.755, -17.051, -84.401, 50.679]
  Set speed (120.0 mm/s)
  MoveL 1485 to (490.4, 509.6, 2.8) mm, rotated rx 0 ry 90 rz 0 deg; joints [-13.088, -26.71, 111.769, -17.069, -84.413, 50.677]
  Set speed (15.0 mm/s)
  Call Extruder(0.559)
  MoveL 1486 to (490.4, 490.4, 2.8) mm, rotated rx 0 ry 90 rz 0 deg; joints [-11.303, -26.775, 112.257, -15.265, -84.779, 50.417]
  MoveL 1487 to (509.6, 490.4, 2.8) mm, rotated rx 0 ry 90 rz 0 deg; joints [-10.955, -26.446, 109.971, -14.97, -82.88, 50.898]
  MoveL 1488 to (509.6, 509.6, 2.8) mm, rotated rx 0 ry 90 rz 0 deg; joints [-12.688, -26.37, 109.487, -16.731, -82.544, 51.205]
  MoveL 1489 to (490.4, 509.6, 2.8) mm, rotated rx 0 ry 90 rz 0 deg; joints [-13.088, -26.71, 111.769, -17.069, -84.413, 50.677]
  Set speed (120.0 mm/s)
  MoveL 1490 to (490.4, 509.2, 2.8) mm, rotated rx 0 ry 90 rz 0 deg; joints [-13.051, -26.711, 111.78, -17.031, -84.421, 50.671]
  Set speed (1000.0 mm/s)
  MoveL 1491 to (491.1, 508.9, 2.8) mm, rotated rx 0 ry 90 rz 0 deg; joints [-13.008, -26.701, 111.705, -16.99, -84.359, 50.686]
  Set speed (1000.0 mm/s)
  MoveL 1492 to (490.68, 490.68, 2.8) mm, rotated rx 0 ry 90 rz 0 deg; joints [-11.324, -26.77, 112.218, -15.287, -84.746, 50.427]
  Set speed (1000.0 mm/s)
  MoveL 1493 to (490.68, 490.68, 2.9) mm, rotated rx 0 ry 90 rz 0 deg; joints [-11.324, -26.781, 112.223, -15.287, -84.741, 50.429]
  Set speed (30.0 mm/s)
  Call Extruder(0.767)
  MoveL 1494 to (509.32, 509.32, 2.9) mm, rotated rx 0 ry 90 rz 0 deg; joints [-12.669, -26.387, 109.534, -16.71, -82.572, 51.194]
  MoveL 1495 to (509.44, 509.44, 2.9) mm, rotated rx 0 ry 90 rz 0 deg; joints [-12.677, -26.384, 109.516, -16.719, -82.558, 51.2]
  Set speed (120.0 mm/s)
  MoveL 1496 to (509.32, 500.58, 2.9) mm, rotated rx 0 ry 90 rz 0 deg; joints [-11.882, -26.423, 109.763, -15.91, -82.73, 51.05]
  Set speed (30.0 mm/s)
  Call Extruder(0.360)
  MoveL 1497 to (500.58, 509.32, 2.9) mm, rotated rx 0 ry 90 rz 0 deg; joints [-12.847, -26.549, 110.578, -16.859, -83.422, 50.957]
  Set speed (120.0 mm/s)
  MoveL 1498 to (499.42, 509.32, 2.9) mm, rotated rx 0 ry 90 rz 0 deg; joints [-12.872, -26.57, 110.716, -16.879, -83.535, 50.925]
  Set speed (30.0 mm/s)
  Call Extruder(0.360)
  MoveL 1499 to (490.68, 500.58, 2.9) mm, rotated rx 0 ry 90 rz 0 deg; joints [-12.247, -26.748, 111.98, -16.219, -84.558, 50.559]
  Set speed (120.0 mm/s)
  MoveL 1500 to (490.68, 499.42, 2.9) mm, rotated rx 0 ry 90 rz 0 deg; joints [-12.139, -26.752, 112.009, -16.11, -84.58, 50.543]
  Set speed (30.0 mm/s)
  MoveL 1501 to (499.42, 490.68, 2.9) mm, rotated rx 0 ry 90 rz 0 deg; joints [-11.163, -26.638, 111.188, -15.148, -83.876, 50.65]
  Set speed (120.0 mm/s)
  MoveL 1502 to (500.58, 490.68, 2.9) mm, rotated rx 0 ry 90 rz 0 deg; joints [-11.141, -26.618, 111.05, -15.13, -83.761, 50.68]
  Set speed (30.0 mm/s)
  Call Extruder(0.360)
  MoveL 1503 to (509.32, 499.42, 2.9) mm, rotated rx 0 ry 90 rz 0 deg; joints [-11.777, -26.428, 109.792, -15.804, -82.75, 51.032]
  MoveL 1504 to (509.44, 499.54, 2.9) mm, rotated rx 0 ry 90 rz 0 deg; joints [-11.786, -26.425, 109.774, -15.813, -82.736, 51.037]
  Set speed (120.0 mm/s)
  MoveL 1505 to (509.32, 490.68, 2.9) mm, rotated rx 0 ry 90 rz 0 deg; joints [-10.985, -26.461, 110.003, -15, -82.898, 50.896]
  Set speed (30.0 mm/s)
  Call Extruder(0.767)
  MoveL 1506 to (490.68, 509.32, 2.9) mm, rotated rx 0 ry 90 rz 0 deg; joints [-13.056, -26.717, 111.749, -17.037, -84.387, 50.682]
  MoveL 1507 to (490.56, 509.44, 2.9) mm, rotated rx 0 ry 90 rz 0 deg; joints [-13.07, -26.719, 111.76, -17.051, -84.396, 50.68]
  Set speed (120.0 mm/s)
  MoveL 1508 to (490.4, 509.6, 2.9) mm, rotated rx 0 ry 90 rz 0 deg; joints [-13.088, -26.72, 111.774, -17.069, -84.408, 50.678]
  Set speed (15.0 mm/s)
  Call Extruder(0.559)
  MoveL 1509 to (490.4, 490.4, 2.9) mm, rotated rx 0 ry 90 rz 0 deg; joints [-11.303, -26.786, 112.263, -15.265, -84.773, 50.418]
  MoveL 1510 to (509.6, 490.4, 2.9) mm, rotated rx 0 ry 90 rz 0 deg; joints [-10.955, -26.457, 109.976, -14.97, -82.875, 50.899]
  MoveL 1511 to (509.6, 509.6, 2.9) mm, rotated rx 0 ry 90 rz 0 deg; joints [-12.688, -26.38, 109.493, -16.731, -82.539, 51.207]
  MoveL 1512 to (490.4, 509.6, 2.9) mm, rotated rx 0 ry 90 rz 0 deg; joints [-13.088, -26.72, 111.774, -17.069, -84.408, 50.678]
  Set speed (120.0 mm/s)
  MoveL 1513 to (490.4, 509.2, 2.9) mm, rotated rx 0 ry 90 rz 0 deg; joints [-13.051, -26.722, 111.785, -17.031, -84.416, 50.673]
  Set speed (1000.0 mm/s)
  MoveL 1514 to (491.1, 508.9, 2.9) mm, rotated rx 0 ry 90 rz 0 deg; joints [-13.008, -26.712, 111.711, -16.99, -84.354, 50.688]
  Set speed (1000.0 mm/s)
  MoveL 1515 to (490.68, 490.68, 2.9) mm, rotated rx 0 ry 90 rz 0 deg; joints [-11.324, -26.781, 112.223, -15.287, -84.741, 50.429]
  Set speed (1000.0 mm/s)
  MoveL 1516 to (490.68, 490.68, 3) mm, rotated rx 0 ry 90 rz 0 deg; joints [-11.324, -26.791, 112.229, -15.287, -84.736, 50.43]
  Set speed (30.0 mm/s)
  Call Extruder(0.767)
  MoveL 1517 to (509.32, 509.32, 3) mm, rotated rx 0 ry 90 rz 0 deg; joints [-12.669, -26.397, 109.539, -16.71, -82.567, 51.196]
  MoveL 1518 to (509.44, 509.44, 3) mm, rotated rx 0 ry 90 rz 0 deg; joints [-12.677, -26.394, 109.521, -16.719, -82.553, 51.201]
  Set speed (120.0 mm/s)
  MoveL 1519 to (509.11, 500.79, 3) mm, rotated rx 0 ry 90 rz 0 deg; joints [-11.905, -26.437, 109.788, -15.933, -82.742, 51.05]
  Set speed (30.0 mm/s)
  Call Extruder(0.351)
  MoveL 1520 to (500.58, 509.32, 3) mm, rotated rx 0 ry 90 rz 0 deg; joints [-12.847, -26.56, 110.584, -16.859, -83.417, 50.958]
  Set speed (120.0 mm/s)
  MoveL 1521 to (499.42, 509.32, 3) mm, rotated rx 0 ry 90 rz 0 deg; joints [-12.872, -26.58, 110.722, -16.879, -83.53, 50.927]
  Set speed (30.0 mm/s)
  Call Extruder(0.360)
  MoveL 1522 to (490.68, 500.58, 3) mm, rotated rx 0 ry 90 rz 0 deg; joints [-12.247, -26.759, 111.985, -16.219, -84.553, 50.56]
  Set speed (120.0 mm/s)
  MoveL 1523 to (490.68, 499.42, 3) mm, rotated rx 0 ry 90 rz 0 deg; joints [-12.139, -26.763, 112.015, -16.11, -84.575, 50.544]
  Set speed (30.0 mm/s)
  MoveL 1524 to (499.42, 490.68, 3) mm, rotated rx 0 ry 90 rz 0 deg; joints [-11.163, -26.649, 111.193, -15.148, -83.871, 50.652]
  Set speed (120.0 mm/s)
  MoveL 1525 to (500.58, 490.68, 3) mm, rotated rx 0 ry 90 rz 0 deg; joints [-11.141, -26.629, 111.055, -15.131, -83.756, 50.681]
  Set speed (30.0 mm/s)
  Call Extruder(0.324)
  MoveL 1526 to (508.45, 498.55, 3) mm, rotated rx 0 ry 90 rz 0 deg; joints [-11.715, -26.458, 109.924, -15.737, -82.846, 50.997]
  MoveL 1527 to (508.57, 498.67, 3) mm, rotated rx 0 ry 90 rz 0 deg; joints [-11.723, -26.455, 109.906, -15.747, -82.832, 51.002]
  Set speed (120.0 mm/s)
  MoveL 1528 to (509.32, 490.68, 3) mm, rotated rx 0 ry 90 rz 0 deg; joints [-10.985, -26.471, 110.009, -15, -82.893, 50.898]
  Set speed (30.0 mm/s)
  Call Extruder(0.767)
  MoveL 1529 to (490.68, 509.32, 3) mm, rotated rx 0 ry 90 rz 0 deg; joints [-13.056, -26.728, 111.754, -17.037, -84.382, 50.684]
  MoveL 1530 to (490.56, 509.44, 3) mm, rotated rx 0 ry 90 rz 0 deg; joints [-13.07, -26.729, 111.765, -17.051, -84.391, 50.682]
  Set speed (120.0 mm/s)
  MoveL 1531 to (490.4, 509.6, 3) mm, rotated rx 0 ry 90 rz 0 deg; joints [-13.088, -26.731, 111.779, -17.069, -84.403, 50.68]
  Set speed (15.0 mm/s)
  Call Extruder(0.559)
  MoveL 1532 to (490.4, 490.4, 3) mm, rotated rx 0 ry 90 rz 0 deg; joints [-11.303, -26.797, 112.268, -15.265, -84.768, 50.419]
  MoveL 1533 to (509.6, 490.4, 3) mm, rotated rx 0 ry 90 rz 0 deg; joints [-10.955, -26.467, 109.981, -14.971, -82.87, 50.9]
  MoveL 1534 to (509.6, 509.6, 3) mm, rotated rx 0 ry 90 rz 0 deg; joints [-12.688, -26.39, 109.498, -16.731, -82.534, 51.208]
  MoveL 1535 to (490.4, 509.6, 3) mm, rotated rx 0 ry 90 rz 0 deg; joints [-13.088, -26.731, 111.779, -17.069, -84.403, 50.68]
  Set speed (120.0 mm/s)
  MoveL 1536 to (490.4, 509.2, 3) mm, rotated rx 0 ry 90 rz 0 deg; joints [-13.051, -26.733, 111.79, -17.031, -84.411, 50.674]
  Set speed (1000.0 mm/s)
  MoveL 1537 to (490.5, 509.2, 3) mm, rotated rx 0 ry 90 rz 0 deg; joints [-13.049, -26.731, 111.779, -17.03, -84.401, 50.677]
  Set speed (1000.0 mm/s)
  MoveL 1538 to (494.72, 492.25, 3) mm, rotated rx 0 ry 90 rz 0 deg; joints [-11.395, -26.722, 111.714, -15.37, -84.308, 50.554]
  Set speed (15.0 mm/s)
  Call Extruder(0.034)
  MoveL 1539 to (494.72, 491.09, 3) mm, rotated rx 0 ry 90 rz 0 deg; joints [-11.287, -26.726, 111.742, -15.261, -84.328, 50.539]
  Call Extruder(0.068)
  MoveL 1540 to (497.04, 491.09, 3) mm, rotated rx 0 ry 90 rz 0 deg; joints [-11.244, -26.688, 111.466, -15.224, -84.098, 50.598]
  Call Extruder(0.034)
  MoveL 1541 to (497.03, 492.25, 3) mm, rotated rx 0 ry 90 rz 0 deg; joints [-11.352, -26.684, 111.44, -15.333, -84.079, 50.613]
  Call Extruder(0.067)
  MoveL 1542 to (494.72, 492.25, 3) mm, rotated rx 0 ry 90 rz 0 deg; joints [-11.395, -26.722, 111.714, -15.37, -84.308, 50.554]
  Set speed (120.0 mm/s)
  MoveL 1543 to (495.04, 491.94, 3) mm, rotated rx 0 ry 90 rz 0 deg; joints [-11.36, -26.718, 111.683, -15.335, -84.281, 50.558]
  Set speed (15.0 mm/s)
  Call Extruder(0.022)
  MoveL 1544 to (495.58, 491.4, 3) mm, rotated rx 0 ry 90 rz 0 deg; joints [-11.3, -26.711, 111.633, -15.277, -84.238, 50.565]
  Set speed (120.0 mm/s)
  MoveL 1545 to (496.03, 491.94, 3) mm, rotated rx 0 ry 90 rz 0 deg; joints [-11.341, -26.702, 111.566, -15.319, -84.184, 50.583]
  Set speed (15.0 mm/s)
  MoveL 1546 to (496.57, 491.4, 3) mm, rotated rx 0 ry 90 rz 0 deg; joints [-11.282, -26.695, 111.515, -15.261, -84.14, 50.59]
  Set speed (120.0 mm/s)
  MoveL 1547 to (502.13, 491.09, 3) mm, rotated rx 0 ry 90 rz 0 deg; joints [-11.151, -26.601, 110.86, -15.145, -83.596, 50.726]
  Set speed (15.0 mm/s)
  Call Extruder(0.073)
  MoveL 1548 to (504.63, 491.09, 3) mm, rotated rx 0 ry 90 rz 0 deg; joints [-11.106, -26.556, 110.562, -15.107, -83.349, 50.788]
  Call Extruder(0.034)
  MoveL 1549 to (504.63, 492.25, 3) mm, rotated rx 0 ry 90 rz 0 deg; joints [-11.212, -26.552, 110.534, -15.215, -83.329, 50.805]
  Call Extruder(0.073)
  MoveL 1550 to (502.13, 492.25, 3) mm, rotated rx 0 ry 90 rz 0 deg; joints [-11.258, -26.597, 110.833, -15.253, -83.576, 50.742]
  Call Extruder(0.034)
  MoveL 1551 to (502.13, 491.09, 3) mm, rotated rx 0 ry 90 rz 0 deg; joints [-11.151, -26.601, 110.86, -15.145, -83.596, 50.726]
  Set speed (120.0 mm/s)
  MoveL 1552 to (502.96, 491.94, 3) mm, rotated rx 0 ry 90 rz 0 deg; joints [-11.214, -26.583, 110.741, -15.211, -83.499, 50.758]
  Set speed (15.0 mm/s)
  Call Extruder(0.022)
  MoveL 1553 to (503.49, 491.4, 3) mm, rotated rx 0 ry 90 rz 0 deg; joints [-11.155, -26.575, 110.69, -15.154, -83.456, 50.764]
  Set speed (120.0 mm/s)
  MoveL 1554 to (503.95, 491.94, 3) mm, rotated rx 0 ry 90 rz 0 deg; joints [-11.196, -26.565, 110.623, -15.196, -83.402, 50.783]
  Set speed (15.0 mm/s)
  Call Extruder(0.015)
  MoveL 1555 to (504.31, 491.57, 3) mm, rotated rx 0 ry 90 rz 0 deg; joints [-11.156, -26.56, 110.588, -15.157, -83.372, 50.787]
  Set speed (120.0 mm/s)
  MoveL 1556 to (507.72, 498.47, 3) mm, rotated rx 0 ry 90 rz 0 deg; joints [-11.721, -26.472, 110.013, -15.741, -82.919, 50.977]
  Set speed (15.0 mm/s)
  Call Extruder(0.035)
  MoveL 1557 to (508.91, 498.47, 3) mm, rotated rx 0 ry 90 rz 0 deg; joints [-11.699, -26.45, 109.87, -15.723, -82.802, 51.008]
  Call Extruder(0.070)
  MoveL 1558 to (508.91, 500.87, 3) mm, rotated rx 0 ry 90 rz 0 deg; joints [-11.916, -26.44, 109.81, -15.943, -82.76, 51.046]
  Call Extruder(0.035)
  MoveL 1559 to (507.69, 500.87, 3) mm, rotated rx 0 ry 90 rz 0 deg; joints [-11.939, -26.463, 109.956, -15.963, -82.879, 51.014]
  Call Extruder(0.070)
  MoveL 1560 to (507.72, 498.47, 3) mm, rotated rx 0 ry 90 rz 0 deg; joints [-11.721, -26.472, 110.013, -15.741, -82.919, 50.977]
  Set speed (120.0 mm/s)
  MoveL 1561 to (508.59, 499.17, 3) mm, rotated rx 0 ry 90 rz 0 deg; joints [-11.769, -26.453, 109.89, -15.793, -82.821, 51.011]
  Set speed (15.0 mm/s)
  Call Extruder(0.024)
  MoveL 1562 to (508.02, 499.75, 3) mm, rotated rx 0 ry 90 rz 0 deg; joints [-11.832, -26.461, 109.945, -15.855, -82.867, 51.005]
  Set speed (120.0 mm/s)
  MoveL 1563 to (508.59, 500.16, 3) mm, rotated rx 0 ry 90 rz 0 deg; joints [-11.858, -26.449, 109.865, -15.884, -82.803, 51.026]
  Set speed (15.0 mm/s)
  Call Extruder(0.016)
  MoveL 1564 to (508.2, 500.55, 3) mm, rotated rx 0 ry 90 rz 0 deg; joints [-11.901, -26.455, 109.902, -15.926, -82.835, 51.022]
  Set speed (120.0 mm/s)
  MoveL 1565 to (490.68, 490.68, 3) mm, rotated rx 0 ry 90 rz 0 deg; joints [-11.324, -26.791, 112.229, -15.287, -84.736, 50.43]
  Set speed (1000.0 mm/s)
  MoveL 1566 to (490.68, 490.68, 3.1) mm, rotated rx 0 ry 90 rz 0 deg; joints [-11.324, -26.802, 112.234, -15.287, -84.731, 50.431]
  Set speed (30.0 mm/s)
  Call Extruder(0.767)
  MoveL 1567 to (509.32, 509.32, 3.1) mm, rotated rx 0 ry 90 rz 0 deg; joints [-12.669, -26.407, 109.545, -16.71, -82.562, 51.197]
  MoveL 1568 to (509.44, 509.44, 3.1) mm, rotated rx 0 ry 90 rz 0 deg; joints [-12.677, -26.405, 109.527, -16.72, -82.548, 51.203]
  Set speed (120.0 mm/s)
  MoveL 1569 to (509.11, 500.79, 3.1) mm, rotated rx 0 ry 90 rz 0 deg; joints [-11.905, -26.447, 109.793, -15.933, -82.737, 51.051]
  Set speed (30.0 mm/s)
  Call Extruder(0.351)
  MoveL 1570 to (500.58, 509.32, 3.1) mm, rotated rx 0 ry 90 rz 0 deg; joints [-12.847, -26.57, 110.589, -16.859, -83.412, 50.96]
  Set speed (120.0 mm/s)
  MoveL 1571 to (499.42, 509.32, 3.1) mm, rotated rx 0 ry 90 rz 0 deg; joints [-12.872, -26.591, 110.727, -16.879, -83.525, 50.928]
  Set speed (30.0 mm/s)
  Call Extruder(0.360)
  MoveL 1572 to (490.68, 500.58, 3.1) mm, rotated rx 0 ry 90 rz 0 deg; joints [-12.247, -26.77, 111.991, -16.219, -84.548, 50.562]
  Set speed (120.0 mm/s)
  MoveL 1573 to (490.68, 499.42, 3.1) mm, rotated rx 0 ry 90 rz 0 deg; joints [-12.139, -26.774, 112.02, -16.11, -84.57, 50.546]
  Set speed (30.0 mm/s)
  MoveL 1574 to (499.42, 490.68, 3.1) mm, rotated rx 0 ry 90 rz 0 deg; joints [-11.163, -26.66, 111.199, -15.149, -83.866, 50.653]
  Set speed (120.0 mm/s)
  MoveL 1575 to (500.58, 490.68, 3.1) mm, rotated rx 0 ry 90 rz 0 deg; joints [-11.142, -26.64, 111.061, -15.131, -83.751, 50.682]
  Set speed (30.0 mm/s)
  Call Extruder(0.324)
  MoveL 1576 to (508.45, 498.55, 3.1) mm, rotated rx 0 ry 90 rz 0 deg; joints [-11.715, -26.469, 109.929, -15.738, -82.841, 50.998]
  MoveL 1577 to (508.57, 498.67, 3.1) mm, rotated rx 0 ry 90 rz 0 deg; joints [-11.723, -26.466, 109.911, -15.747, -82.827, 51.003]
  Set speed (120.0 mm/s)
  MoveL 1578 to (509.32, 490.68, 3.1) mm, rotated rx 0 ry 90 rz 0 deg; joints [-10.985, -26.482, 110.014, -15.001, -82.888, 50.899]
  Set speed (30.0 mm/s)
  Call Extruder(0.767)
  MoveL 1579 to (490.68, 509.32, 3.1) mm, rotated rx 0 ry 90 rz 0 deg; joints [-13.056, -26.738, 111.76, -17.038, -84.377, 50.685]
  MoveL 1580 to (490.56, 509.44, 3.1) mm, rotated rx 0 ry 90 rz 0 deg; joints [-13.07, -26.74, 111.771, -17.051, -84.386, 50.684]
  Set speed (120.0 mm/s)
  MoveL 1581 to (490.4, 509.6, 3.1) mm, rotated rx 0 ry 90 rz 0 deg; joints [-13.088, -26.742, 111.785, -17.069, -84.398, 50.681]
  Set speed (15.0 mm/s)
  Call Extruder(0.559)
  MoveL 1582 to (490.4, 490.4, 3.1) mm, rotated rx 0 ry 90 rz 0 deg; joints [-11.303, -26.807, 112.273, -15.266, -84.763, 50.421]
  MoveL 1583 to (509.6, 490.4, 3.1) mm, rotated rx 0 ry 90 rz 0 deg; joints [-10.955, -26.478, 109.987, -14.971, -82.865, 50.902]
  MoveL 1584 to (509.6, 509.6, 3.1) mm, rotated rx 0 ry 90 rz 0 deg; joints [-12.688, -26.401, 109.503, -16.731, -82.529, 51.21]
  MoveL 1585 to (490.4, 509.6, 3.1) mm, rotated rx 0 ry 90 rz 0 deg; joints [-13.088, -26.742, 111.785, -17.069, -84.398, 50.681]
  Set speed (120.0 mm/s)
  MoveL 1586 to (490.4, 509.2, 3.1) mm, rotated rx 0 ry 90 rz 0 deg; joints [-13.051, -26.743, 111.796, -17.032, -84.406, 50.676]
  Set speed (1000.0 mm/s)
  MoveL 1587 to (490.5, 509.2, 3.1) mm, rotated rx 0 ry 90 rz 0 deg; joints [-13.049, -26.742, 111.784, -17.03, -84.396, 50.678]
  Set speed (1000.0 mm/s)
  MoveL 1588 to (494.72, 492.25, 3.1) mm, rotated rx 0 ry 90 rz 0 deg; joints [-11.395, -26.733, 111.719, -15.37, -84.303, 50.555]
  Set speed (15.0 mm/s)
  Call Extruder(0.034)
  MoveL 1589 to (494.72, 491.09, 3.1) mm, rotated rx 0 ry 90 rz 0 deg; joints [-11.287, -26.737, 111.747, -15.261, -84.323, 50.54]
  Call Extruder(0.070)
  MoveL 1590 to (497.11, 491.09, 3.1) mm, rotated rx 0 ry 90 rz 0 deg; joints [-11.243, -26.697, 111.463, -15.223, -84.086, 50.601]
  Call Extruder(0.034)
  MoveL 1591 to (497.11, 492.25, 3.1) mm, rotated rx 0 ry 90 rz 0 deg; joints [-11.35, -26.693, 111.435, -15.332, -84.066, 50.617]
  Call Extruder(0.070)
  MoveL 1592 to (494.72, 492.25, 3.1) mm, rotated rx 0 ry 90 rz 0 deg; joints [-11.395, -26.733, 111.719, -15.37, -84.303, 50.555]
  Set speed (120.0 mm/s)
  MoveL 1593 to (495.37, 491.41, 3.1) mm, rotated rx 0 ry 90 rz 0 deg; joints [-11.304, -26.725, 111.663, -15.28, -84.254, 50.561]
  Set speed (15.0 mm/s)
  Call Extruder(0.022)
  MoveL 1594 to (495.9, 491.94, 3.1) mm, rotated rx 0 ry 90 rz 0 deg; joints [-11.344, -26.714, 111.587, -15.321, -84.192, 50.581]
  Set speed (120.0 mm/s)
  MoveL 1595 to (496.36, 491.4, 3.1) mm, rotated rx 0 ry 90 rz 0 deg; joints [-11.286, -26.709, 111.546, -15.264, -84.156, 50.586]
  Set speed (15.0 mm/s)
  Call Extruder(0.018)
  MoveL 1596 to (496.8, 491.85, 3.1) mm, rotated rx 0 ry 90 rz 0 deg; joints [-11.319, -26.7, 111.483, -15.299, -84.104, 50.603]
  Set speed (120.0 mm/s)
  MoveL 1597 to (502.07, 492.25, 3.1) mm, rotated rx 0 ry 90 rz 0 deg; joints [-11.259, -26.608, 110.846, -15.254, -83.577, 50.742]
  Set speed (15.0 mm/s)
  Call Extruder(0.034)
  MoveL 1598 to (502.07, 491.09, 3.1) mm, rotated rx 0 ry 90 rz 0 deg; joints [-11.152, -26.612, 110.873, -15.146, -83.597, 50.725]
  Call Extruder(0.075)
  MoveL 1599 to (504.63, 491.09, 3.1) mm, rotated rx 0 ry 90 rz 0 deg; joints [-11.106, -26.567, 110.567, -15.108, -83.344, 50.789]
  Call Extruder(0.034)
  MoveL 1600 to (504.63, 492.25, 3.1) mm, rotated rx 0 ry 90 rz 0 deg; joints [-11.212, -26.563, 110.54, -15.215, -83.324, 50.806]
  Call Extruder(0.075)
  MoveL 1601 to (502.07, 492.25, 3.1) mm, rotated rx 0 ry 90 rz 0 deg; joints [-11.259, -26.608, 110.846, -15.254, -83.577, 50.742]
  Set speed (120.0 mm/s)
  MoveL 1602 to (502.83, 491.94, 3.1) mm, rotated rx 0 ry 90 rz 0 deg; joints [-11.216, -26.596, 110.763, -15.213, -83.508, 50.756]
  Set speed (15.0 mm/s)
  Call Extruder(0.018)
  MoveL 1603 to (502.38, 491.49, 3.1) mm, rotated rx 0 ry 90 rz 0 deg; joints [-11.184, -26.605, 110.826, -15.179, -83.559, 50.739]
  Set speed (120.0 mm/s)
  MoveL 1604 to (503.28, 491.4, 3.1) mm, rotated rx 0 ry 90 rz 0 deg; joints [-11.159, -26.59, 110.721, -15.157, -83.471, 50.76]
  Set speed (15.0 mm/s)
  Call Extruder(0.022)
  MoveL 1605 to (503.82, 491.94, 3.1) mm, rotated rx 0 ry 90 rz 0 deg; joints [-11.198, -26.578, 110.644, -15.198, -83.41, 50.781]
  Set speed (120.0 mm/s)
  MoveL 1606 to (507.69, 498.47, 3.1) mm, rotated rx 0 ry 90 rz 0 deg; joints [-11.721, -26.483, 110.021, -15.742, -82.916, 50.978]
  Set speed (15.0 mm/s)
  Call Extruder(0.035)
  MoveL 1607 to (508.91, 498.47, 3.1) mm, rotated rx 0 ry 90 rz 0 deg; joints [-11.699, -26.46, 109.875, -15.723, -82.797, 51.009]
  Call Extruder(0.070)
  MoveL 1608 to (508.91, 500.87, 3.1) mm, rotated rx 0 ry 90 rz 0 deg; joints [-11.916, -26.451, 109.815, -15.944, -82.755, 51.047]
  Call Extruder(0.035)
  MoveL 1609 to (507.7, 500.87, 3.1) mm, rotated rx 0 ry 90 rz 0 deg; joints [-11.939, -26.474, 109.961, -15.963, -82.874, 51.016]
  Call Extruder(0.070)
  MoveL 1610 to (507.69, 498.47, 3.1) mm, rotated rx 0 ry 90 rz 0 deg; joints [-11.721, -26.483, 110.021, -15.742, -82.916, 50.978]
  Set speed (120.0 mm/s)
  MoveL 1611 to (508.01, 499.1, 3.1) mm, rotated rx 0 ry 90 rz 0 deg; joints [-11.773, -26.475, 109.968, -15.795, -82.874, 50.996]
  Set speed (15.0 mm/s)
  Call Extruder(0.024)
  MoveL 1612 to (508.59, 499.68, 3.1) mm, rotated rx 0 ry 90 rz 0 deg; joints [-11.815, -26.461, 109.883, -15.84, -82.807, 51.02]
  Set speed (120.0 mm/s)
  MoveL 1613 to (508.01, 500.09, 3.1) mm, rotated rx 0 ry 90 rz 0 deg; joints [-11.863, -26.471, 109.943, -15.886, -82.857, 51.011]
  Set speed (15.0 mm/s)
  Call Extruder(0.019)
  MoveL 1614 to (508.47, 500.55, 3.1) mm, rotated rx 0 ry 90 rz 0 deg; joints [-11.896, -26.46, 109.875, -15.922, -82.803, 51.031]
  Set speed (120.0 mm/s)
  MoveL 1615 to (490.68, 490.68, 3.1) mm, rotated rx 0 ry 90 rz 0 deg; joints [-11.324, -26.802, 112.234, -15.287, -84.731, 50.431]
  Set speed (1000.0 mm/s)
  MoveL 1616 to (490.68, 490.68, 3.2) mm, rotated rx 0 ry 90 rz 0 deg; joints [-11.324, -26.813, 112.239, -15.287, -84.726, 50.433]
  Set speed (30.0 mm/s)
  Call Extruder(0.767)
  MoveL 1617 to (509.32, 509.32, 3.2) mm, rotated rx 0 ry 90 rz 0 deg; joints [-12.669, -26.418, 109.55, -16.711, -82.557, 51.199]
  MoveL 1618 to (509.44, 509.44, 3.2) mm, rotated rx 0 ry 90 rz 0 deg; joints [-12.677, -26.415, 109.532, -16.72, -82.543, 51.204]
  Set speed (120.0 mm/s)
  MoveL 1619 to (509.11, 500.79, 3.2) mm, rotated rx 0 ry 90 rz 0 deg; joints [-11.905, -26.458, 109.798, -15.933, -82.732, 51.052]
  Set speed (30.0 mm/s)
  Call Extruder(0.351)
  MoveL 1620 to (500.58, 509.32, 3.2) mm, rotated rx 0 ry 90 rz 0 deg; joints [-12.847, -26.581, 110.594, -16.859, -83.407, 50.961]
  Set speed (120.0 mm/s)
  MoveL 1621 to (499.42, 509.32, 3.2) mm, rotated rx 0 ry 90 rz 0 deg; joints [-12.872, -26.601, 110.732, -16.88, -83.52, 50.93]
  Set speed (30.0 mm/s)
  Call Extruder(0.360)
  MoveL 1622 to (490.68, 500.58, 3.2) mm, rotated rx 0 ry 90 rz 0 deg; joints [-12.247, -26.78, 111.996, -16.219, -84.543, 50.563]
  Set speed (120.0 mm/s)
  MoveL 1623 to (490.68, 499.42, 3.2) mm, rotated rx 0 ry 90 rz 0 deg; joints [-12.139, -26.784, 112.025, -16.11, -84.565, 50.547]
  Set speed (30.0 mm/s)
  MoveL 1624 to (499.42, 490.68, 3.2) mm, rotated rx 0 ry 90 rz 0 deg; joints [-11.163, -26.67, 111.204, -15.149, -83.861, 50.655]
  Set speed (120.0 mm/s)
  MoveL 1625 to (500.58, 490.68, 3.2) mm, rotated rx 0 ry 90 rz 0 deg; joints [-11.141, -26.65, 111.066, -15.131, -83.746, 50.684]
  Set speed (30.0 mm/s)
  Call Extruder(0.324)
  MoveL 1626 to (508.44, 498.54, 3.2) mm, rotated rx 0 ry 90 rz 0 deg; joints [-11.714, -26.479, 109.935, -15.738, -82.836, 51]
  MoveL 1627 to (508.57, 498.67, 3.2) mm, rotated rx 0 ry 90 rz 0 deg; joints [-11.723, -26.476, 109.917, -15.747, -82.822, 51.005]
  Set speed (120.0 mm/s)
  MoveL 1628 to (509.32, 490.68, 3.2) mm, rotated rx 0 ry 90 rz 0 deg; joints [-10.985, -26.492, 110.019, -15.001, -82.883, 50.9]
  Set speed (30.0 mm/s)
  Call Extruder(0.767)
  MoveL 1629 to (490.68, 509.32, 3.2) mm, rotated rx 0 ry 90 rz 0 deg; joints [-13.056, -26.749, 111.765, -17.038, -84.372, 50.687]
  MoveL 1630 to (490.56, 509.44, 3.2) mm, rotated rx 0 ry 90 rz 0 deg; joints [-13.07, -26.75, 111.776, -17.051, -84.381, 50.685]
  Set speed (120.0 mm/s)
  MoveL 1631 to (490.4, 509.6, 3.2) mm, rotated rx 0 ry 90 rz 0 deg; joints [-13.088, -26.752, 111.79, -17.069, -84.393, 50.683]
  Set speed (15.0 mm/s)
  Call Extruder(0.559)
  MoveL 1632 to (490.4, 490.4, 3.2) mm, rotated rx 0 ry 90 rz 0 deg; joints [-11.303, -26.818, 112.279, -15.266, -84.758, 50.422]
  MoveL 1633 to (509.6, 490.4, 3.2) mm, rotated rx 0 ry 90 rz 0 deg; joints [-10.955, -26.488, 109.992, -14.971, -82.86, 50.903]
  MoveL 1634 to (509.6, 509.6, 3.2) mm, rotated rx 0 ry 90 rz 0 deg; joints [-12.688, -26.411, 109.509, -16.732, -82.525, 51.211]
  MoveL 1635 to (490.4, 509.6, 3.2) mm, rotated rx 0 ry 90 rz 0 deg; joints [-13.088, -26.752, 111.79, -17.069, -84.393, 50.683]
  Set speed (120.0 mm/s)
  MoveL 1636 to (490.4, 509.2, 3.2) mm, rotated rx 0 ry 90 rz 0 deg; joints [-13.051, -26.754, 111.801, -17.032, -84.401, 50.677]
  Set speed (1000.0 mm/s)
  MoveL 1637 to (490.5, 509.2, 3.2) mm, rotated rx 0 ry 90 rz 0 deg; joints [-13.049, -26.752, 111.789, -17.03, -84.391, 50.68]
  Set speed (1000.0 mm/s)
  MoveL 1638 to (494.72, 492.25, 3.2) mm, rotated rx 0 ry 90 rz 0 deg; joints [-11.395, -26.743, 111.724, -15.37, -84.298, 50.557]
  Set speed (15.0 mm/s)
  Call Extruder(0.034)
  MoveL 1639 to (494.72, 491.09, 3.2) mm, rotated rx 0 ry 90 rz 0 deg; joints [-11.287, -26.747, 111.752, -15.261, -84.318, 50.541]
  Call Extruder(0.071)
  MoveL 1640 to (497.17, 491.09, 3.2) mm, rotated rx 0 ry 90 rz 0 deg; joints [-11.242, -26.707, 111.461, -15.222, -84.075, 50.604]
  Call Extruder(0.034)
  MoveL 1641 to (497.18, 492.25, 3.2) mm, rotated rx 0 ry 90 rz 0 deg; joints [-11.349, -26.703, 111.434, -15.331, -84.055, 50.619]
  Call Extruder(0.071)
  MoveL 1642 to (494.72, 492.25, 3.2) mm, rotated rx 0 ry 90 rz 0 deg; joints [-11.395, -26.743, 111.724, -15.37, -84.298, 50.557]
  Set speed (120.0 mm/s)
  MoveL 1643 to (495.04, 491.94, 3.2) mm, rotated rx 0 ry 90 rz 0 deg; joints [-11.36, -26.739, 111.694, -15.335, -84.271, 50.561]
  Set speed (15.0 mm/s)
  Call Extruder(0.022)
  MoveL 1644 to (495.57, 491.4, 3.2) mm, rotated rx 0 ry 90 rz 0 deg; joints [-11.3, -26.732, 111.644, -15.277, -84.228, 50.567]
  Set speed (120.0 mm/s)
  MoveL 1645 to (496.03, 491.94, 3.2) mm, rotated rx 0 ry 90 rz 0 deg; joints [-11.341, -26.723, 111.577, -15.319, -84.174, 50.586]
  Set speed (15.0 mm/s)
  MoveL 1646 to (496.56, 491.41, 3.2) mm, rotated rx 0 ry 90 rz 0 deg; joints [-11.282, -26.716, 111.526, -15.261, -84.13, 50.592]
  Set speed (120.0 mm/s)
  MoveL 1647 to (502.01, 491.09, 3.2) mm, rotated rx 0 ry 90 rz 0 deg; joints [-11.153, -26.624, 110.886, -15.147, -83.598, 50.725]
  Set speed (15.0 mm/s)
  Call Extruder(0.076)
  MoveL 1648 to (504.63, 491.09, 3.2) mm, rotated rx 0 ry 90 rz 0 deg; joints [-11.106, -26.577, 110.572, -15.108, -83.339, 50.791]
  Call Extruder(0.034)
  MoveL 1649 to (504.63, 492.25, 3.2) mm, rotated rx 0 ry 90 rz 0 deg; joints [-11.212, -26.573, 110.545, -15.215, -83.319, 50.808]
  Call Extruder(0.076)
  MoveL 1650 to (502.01, 492.25, 3.2) mm, rotated rx 0 ry 90 rz 0 deg; joints [-11.26, -26.62, 110.858, -15.255, -83.578, 50.742]
  Call Extruder(0.034)
  MoveL 1651 to (502.01, 491.09, 3.2) mm, rotated rx 0 ry 90 rz 0 deg; joints [-11.153, -26.624, 110.886, -15.147, -83.598, 50.725]
  Set speed (120.0 mm/s)
  MoveL 1652 to (502.5, 491.41, 3.2) mm, rotated rx 0 ry 90 rz 0 deg; joints [-11.173, -26.614, 110.819, -15.169, -83.543, 50.742]
  Set speed (15.0 mm/s)
  Call Extruder(0.007)
  MoveL 1653 to (502.32, 491.59, 3.2) mm, rotated rx 0 ry 90 rz 0 deg; joints [-11.193, -26.617, 110.836, -15.189, -83.558, 50.74]
  Set speed (120.0 mm/s)
  MoveL 1654 to (502.96, 491.94, 3.2) mm, rotated rx 0 ry 90 rz 0 deg; joints [-11.214, -26.604, 110.752, -15.212, -83.489, 50.761]
  Set speed (15.0 mm/s)
  Call Extruder(0.022)
  MoveL 1655 to (503.49, 491.4, 3.2) mm, rotated rx 0 ry 90 rz 0 deg; joints [-11.155, -26.596, 110.701, -15.154, -83.446, 50.767]
  Set speed (120.0 mm/s)
  MoveL 1656 to (503.95, 491.94, 3.2) mm, rotated rx 0 ry 90 rz 0 deg; joints [-11.196, -26.586, 110.634, -15.196, -83.392, 50.786]
  Set speed (15.0 mm/s)
  Call Extruder(0.015)
  MoveL 1657 to (504.31, 491.57, 3.2) mm, rotated rx 0 ry 90 rz 0 deg; joints [-11.156, -26.581, 110.599, -15.157, -83.362, 50.79]
  Set speed (120.0 mm/s)
  MoveL 1658 to (507.7, 498.47, 3.2) mm, rotated rx 0 ry 90 rz 0 deg; joints [-11.721, -26.494, 110.027, -15.742, -82.911, 50.979]
  Set speed (15.0 mm/s)
  Call Extruder(0.035)
  MoveL 1659 to (508.91, 498.47, 3.2) mm, rotated rx 0 ry 90 rz 0 deg; joints [-11.699, -26.471, 109.881, -15.723, -82.792, 51.01]
  Call Extruder(0.070)
  MoveL 1660 to (508.91, 500.87, 3.2) mm, rotated rx 0 ry 90 rz 0 deg; joints [-11.916, -26.461, 109.82, -15.944, -82.75, 51.049]
  Call Extruder(0.035)
  MoveL 1661 to (507.69, 500.87, 3.2) mm, rotated rx 0 ry 90 rz 0 deg; joints [-11.939, -26.484, 109.966, -15.963, -82.869, 51.017]
  Call Extruder(0.070)
  MoveL 1662 to (507.7, 498.47, 3.2) mm, rotated rx 0 ry 90 rz 0 deg; joints [-11.721, -26.494, 110.027, -15.742, -82.911, 50.979]
  Set speed (120.0 mm/s)
  MoveL 1663 to (508.59, 499.17, 3.2) mm, rotated rx 0 ry 90 rz 0 deg; joints [-11.769, -26.474, 109.901, -15.793, -82.811, 51.013]
  Set speed (15.0 mm/s)
  Call Extruder(0.024)
  MoveL 1664 to (508.01, 499.76, 3.2) mm, rotated rx 0 ry 90 rz 0 deg; joints [-11.833, -26.483, 109.957, -15.856, -82.858, 51.008]
  Set speed (120.0 mm/s)
  MoveL 1665 to (508.59, 500.16, 3.2) mm, rotated rx 0 ry 90 rz 0 deg; joints [-11.858, -26.47, 109.876, -15.884, -82.793, 51.029]
  Set speed (15.0 mm/s)
  Call Extruder(0.016)
  MoveL 1666 to (508.2, 500.55, 3.2) mm, rotated rx 0 ry 90 rz 0 deg; joints [-11.901, -26.476, 109.913, -15.926, -82.825, 51.025]
  Set speed (120.0 mm/s)
  MoveL 1667 to (490.68, 490.68, 3.2) mm, rotated rx 0 ry 90 rz 0 deg; joints [-11.324, -26.813, 112.239, -15.287, -84.726, 50.433]
  Set speed (1000.0 mm/s)
  MoveL 1668 to (490.68, 490.68, 3.3) mm, rotated rx 0 ry 90 rz 0 deg; joints [-11.324, -26.823, 112.245, -15.288, -84.72, 50.434]
  Set speed (30.0 mm/s)
  Call Extruder(0.767)
  MoveL 1669 to (509.32, 509.32, 3.3) mm, rotated rx 0 ry 90 rz 0 deg; joints [-12.669, -26.428, 109.555, -16.711, -82.552, 51.2]
  MoveL 1670 to (509.44, 509.44, 3.3) mm, rotated rx 0 ry 90 rz 0 deg; joints [-12.677, -26.425, 109.537, -16.72, -82.538, 51.206]
  Set speed (120.0 mm/s)
  MoveL 1671 to (509.11, 500.79, 3.3) mm, rotated rx 0 ry 90 rz 0 deg; joints [-11.905, -26.468, 109.804, -15.933, -82.727, 51.054]
  Set speed (30.0 mm/s)
  Call Extruder(0.351)
  MoveL 1672 to (500.58, 509.32, 3.3) mm, rotated rx 0 ry 90 rz 0 deg; joints [-12.847, -26.591, 110.6, -16.859, -83.402, 50.963]
  Set speed (120.0 mm/s)
  MoveL 1673 to (499.42, 509.32, 3.3) mm, rotated rx 0 ry 90 rz 0 deg; joints [-12.872, -26.612, 110.738, -16.88, -83.515, 50.931]
  Set speed (30.0 mm/s)
  Call Extruder(0.360)
  MoveL 1674 to (490.68, 500.58, 3.3) mm, rotated rx 0 ry 90 rz 0 deg; joints [-12.247, -26.791, 112.001, -16.219, -84.538, 50.565]
  Set speed (120.0 mm/s)
  MoveL 1675 to (490.68, 499.42, 3.3) mm, rotated rx 0 ry 90 rz 0 deg; joints [-12.139, -26.795, 112.031, -16.111, -84.56, 50.549]
  Set speed (30.0 mm/s)
  MoveL 1676 to (499.42, 490.68, 3.3) mm, rotated rx 0 ry 90 rz 0 deg; joints [-11.163, -26.681, 111.209, -15.149, -83.855, 50.656]
  Set speed (120.0 mm/s)
  MoveL 1677 to (500.58, 490.68, 3.3) mm, rotated rx 0 ry 90 rz 0 deg; joints [-11.141, -26.661, 111.071, -15.131, -83.741, 50.685]
  Set speed (30.0 mm/s)
  Call Extruder(0.060)
  MoveL 1678 to (502.03, 492.13, 3.3) mm, rotated rx 0 ry 90 rz 0 deg; joints [-11.248, -26.63, 110.864, -15.244, -83.573, 50.742]
  Set speed (120.0 mm/s)
  MoveL 1679 to (502.07, 492.17, 3.3) mm, rotated rx 0 ry 90 rz 0 deg; joints [-11.252, -26.63, 110.858, -15.247, -83.568, 50.744]
  Set speed (30.0 mm/s)
  Call Extruder(0.262)
  MoveL 1680 to (508.44, 498.54, 3.3) mm, rotated rx 0 ry 90 rz 0 deg; joints [-11.714, -26.49, 109.94, -15.738, -82.832, 51.001]
  MoveL 1681 to (508.57, 498.67, 3.3) mm, rotated rx 0 ry 90 rz 0 deg; joints [-11.723, -26.487, 109.922, -15.747, -82.817, 51.006]
  Set speed (120.0 mm/s)
  MoveL 1682 to (509.32, 490.68, 3.3) mm, rotated rx 0 ry 90 rz 0 deg; joints [-10.985, -26.503, 110.025, -15.001, -82.878, 50.902]
  Set speed (30.0 mm/s)
  Call Extruder(0.767)
  MoveL 1683 to (490.68, 509.32, 3.3) mm, rotated rx 0 ry 90 rz 0 deg; joints [-13.056, -26.76, 111.77, -17.038, -84.367, 50.688]
  MoveL 1684 to (490.56, 509.44, 3.3) mm, rotated rx 0 ry 90 rz 0 deg; joints [-13.07, -26.761, 111.782, -17.052, -84.376, 50.687]
  Set speed (120.0 mm/s)
  MoveL 1685 to (490.4, 509.6, 3.3) mm, rotated rx 0 ry 90 rz 0 deg; joints [-13.088, -26.763, 111.796, -17.069, -84.388, 50.685]
  Set speed (15.0 mm/s)
  Call Extruder(0.559)
  MoveL 1686 to (490.4, 490.4, 3.3) mm, rotated rx 0 ry 90 rz 0 deg; joints [-11.303, -26.829, 112.284, -15.266, -84.753, 50.424]
  MoveL 1687 to (509.6, 490.4, 3.3) mm, rotated rx 0 ry 90 rz 0 deg; joints [-10.955, -26.499, 109.997, -14.971, -82.855, 50.904]
  MoveL 1688 to (509.6, 509.6, 3.3) mm, rotated rx 0 ry 90 rz 0 deg; joints [-12.688, -26.422, 109.514, -16.732, -82.52, 51.212]
  MoveL 1689 to (490.4, 509.6, 3.3) mm, rotated rx 0 ry 90 rz 0 deg; joints [-13.088, -26.763, 111.796, -17.069, -84.388, 50.685]
  Set speed (120.0 mm/s)
  MoveL 1690 to (490.4, 509.2, 3.3) mm, rotated rx 0 ry 90 rz 0 deg; joints [-13.051, -26.764, 111.807, -17.032, -84.396, 50.679]
  Set speed (1000.0 mm/s)
  MoveL 1691 to (490.5, 509.2, 3.3) mm, rotated rx 0 ry 90 rz 0 deg; joints [-13.049, -26.763, 111.795, -17.03, -84.386, 50.682]
  Set speed (1000.0 mm/s)
  MoveL 1692 to (494.72, 492.25, 3.3) mm, rotated rx 0 ry 90 rz 0 deg; joints [-11.395, -26.754, 111.73, -15.37, -84.292, 50.558]
  Set speed (15.0 mm/s)
  Call Extruder(0.034)
  MoveL 1693 to (494.72, 491.09, 3.3) mm, rotated rx 0 ry 90 rz 0 deg; joints [-11.287, -26.758, 111.758, -15.261, -84.313, 50.543]
  Call Extruder(0.073)
  MoveL 1694 to (497.23, 491.09, 3.3) mm, rotated rx 0 ry 90 rz 0 deg; joints [-11.241, -26.716, 111.46, -15.221, -84.064, 50.606]
  Call Extruder(0.034)
  MoveL 1695 to (497.23, 492.25, 3.3) mm, rotated rx 0 ry 90 rz 0 deg; joints [-11.348, -26.712, 111.432, -15.33, -84.044, 50.622]
  Call Extruder(0.073)
  MoveL 1696 to (494.72, 492.25, 3.3) mm, rotated rx 0 ry 90 rz 0 deg; joints [-11.395, -26.754, 111.73, -15.37, -84.292, 50.558]
  Set speed (120.0 mm/s)
  MoveL 1697 to (495.36, 491.4, 3.3) mm, rotated rx 0 ry 90 rz 0 deg; joints [-11.304, -26.746, 111.674, -15.28, -84.244, 50.563]
  Set speed (15.0 mm/s)
  Call Extruder(0.022)
  MoveL 1698 to (495.9, 491.94, 3.3) mm, rotated rx 0 ry 90 rz 0 deg; joints [-11.344, -26.736, 111.598, -15.322, -84.182, 50.584]
  Set speed (120.0 mm/s)
  MoveL 1699 to (496.35, 491.4, 3.3) mm, rotated rx 0 ry 90 rz 0 deg; joints [-11.286, -26.73, 111.556, -15.265, -84.146, 50.589]
  Set speed (15.0 mm/s)
  MoveL 1700 to (496.89, 491.94, 3.3) mm, rotated rx 0 ry 90 rz 0 deg; joints [-11.325, -26.719, 111.481, -15.306, -84.084, 50.609]
  Set speed (120.0 mm/s)
  MoveL 1701 to (501.95, 492.25, 3.3) mm, rotated rx 0 ry 90 rz 0 deg; joints [-11.261, -26.631, 110.871, -15.256, -83.579, 50.742]
  Set speed (15.0 mm/s)
  Call Extruder(0.034)
  MoveL 1702 to (501.95, 491.09, 3.3) mm, rotated rx 0 ry 90 rz 0 deg; joints [-11.154, -26.635, 110.898, -15.148, -83.599, 50.725]
  Call Extruder(0.078)
  MoveL 1703 to (504.63, 491.09, 3.3) mm, rotated rx 0 ry 90 rz 0 deg; joints [-11.106, -26.588, 110.578, -15.108, -83.334, 50.792]
  Call Extruder(0.034)
  MoveL 1704 to (504.63, 492.25, 3.3) mm, rotated rx 0 ry 90 rz 0 deg; joints [-11.212, -26.584, 110.55, -15.216, -83.314, 50.809]
  Call Extruder(0.078)
  MoveL 1705 to (501.95, 492.25, 3.3) mm, rotated rx 0 ry 90 rz 0 deg; joints [-11.261, -26.631, 110.871, -15.256, -83.579, 50.742]
  Set speed (120.0 mm/s)
  MoveL 1706 to (502.29, 491.41, 3.3) mm, rotated rx 0 ry 90 rz 0 deg; joints [-11.177, -26.628, 110.85, -15.172, -83.559, 50.738]
  Set speed (15.0 mm/s)
  Call Extruder(0.022)
  MoveL 1707 to (502.83, 491.94, 3.3) mm, rotated rx 0 ry 90 rz 0 deg; joints [-11.216, -26.617, 110.773, -15.214, -83.498, 50.759]
  Set speed (120.0 mm/s)
  MoveL 1708 to (503.28, 491.41, 3.3) mm, rotated rx 0 ry 90 rz 0 deg; joints [-11.159, -26.611, 110.731, -15.157, -83.461, 50.763]
  Set speed (15.0 mm/s)
  MoveL 1709 to (503.82, 491.94, 3.3) mm, rotated rx 0 ry 90 rz 0 deg; joints [-11.198, -26.599, 110.655, -15.199, -83.4, 50.784]
  Set speed (120.0 mm/s)
  MoveL 1710 to (507.7, 498.47, 3.3) mm, rotated rx 0 ry 90 rz 0 deg; joints [-11.721, -26.504, 110.032, -15.742, -82.906, 50.981]
  Set speed (15.0 mm/s)
  Call Extruder(0.035)
  MoveL 1711 to (508.91, 498.46, 3.3) mm, rotated rx 0 ry 90 rz 0 deg; joints [-11.698, -26.481, 109.886, -15.723, -82.787, 51.012]
  Call Extruder(0.070)
  MoveL 1712 to (508.91, 500.87, 3.3) mm, rotated rx 0 ry 90 rz 0 deg; joints [-11.916, -26.472, 109.826, -15.944, -82.745, 51.05]
  Call Extruder(0.035)
  MoveL 1713 to (507.69, 500.87, 3.3) mm, rotated rx 0 ry 90 rz 0 deg; joints [-11.939, -26.495, 109.972, -15.963, -82.864, 51.019]
  Call Extruder(0.070)
  MoveL 1714 to (507.7, 498.47, 3.3) mm, rotated rx 0 ry 90 rz 0 deg; joints [-11.721, -26.504, 110.032, -15.742, -82.906, 50.981]
  Set speed (120.0 mm/s)
  MoveL 1715 to (508.01, 499.1, 3.3) mm, rotated rx 0 ry 90 rz 0 deg; joints [-11.773, -26.496, 109.979, -15.796, -82.865, 50.999]
  Set speed (15.0 mm/s)
  Call Extruder(0.024)
  MoveL 1716 to (508.59, 499.68, 3.3) mm, rotated rx 0 ry 90 rz 0 deg; joints [-11.815, -26.482, 109.893, -15.84, -82.797, 51.023]
  Set speed (120.0 mm/s)
  MoveL 1717 to (508.01, 500.09, 3.3) mm, rotated rx 0 ry 90 rz 0 deg; joints [-11.863, -26.492, 109.954, -15.887, -82.847, 51.014]
  Set speed (15.0 mm/s)
  Call Extruder(0.019)
  MoveL 1718 to (508.47, 500.55, 3.3) mm, rotated rx 0 ry 90 rz 0 deg; joints [-11.896, -26.481, 109.886, -15.922, -82.793, 51.034]
  Set speed (120.0 mm/s)
  MoveL 1719 to (490.68, 490.68, 3.3) mm, rotated rx 0 ry 90 rz 0 deg; joints [-11.324, -26.823, 112.245, -15.288, -84.72, 50.434]
  Set speed (1000.0 mm/s)
  MoveL 1720 to (490.68, 490.68, 3.4) mm, rotated rx 0 ry 90 rz 0 deg; joints [-11.324, -26.834, 112.25, -15.288, -84.715, 50.436]
  Set speed (30.0 mm/s)
  Call Extruder(0.767)
  MoveL 1721 to (509.32, 509.32, 3.4) mm, rotated rx 0 ry 90 rz 0 deg; joints [-12.669, -26.439, 109.561, -16.711, -82.547, 51.202]
  MoveL 1722 to (509.44, 509.44, 3.4) mm, rotated rx 0 ry 90 rz 0 deg; joints [-12.677, -26.436, 109.543, -16.72, -82.533, 51.207]
  Set speed (120.0 mm/s)
  MoveL 1723 to (509.11, 500.79, 3.4) mm, rotated rx 0 ry 90 rz 0 deg; joints [-11.905, -26.479, 109.809, -15.934, -82.722, 51.055]
  Set speed (30.0 mm/s)
  Call Extruder(0.351)
  MoveL 1724 to (500.58, 509.32, 3.4) mm, rotated rx 0 ry 90 rz 0 deg; joints [-12.847, -26.602, 110.605, -16.86, -83.397, 50.964]
  Set speed (120.0 mm/s)
  MoveL 1725 to (499.42, 509.32, 3.4) mm, rotated rx 0 ry 90 rz 0 deg; joints [-12.872, -26.622, 110.743, -16.88, -83.51, 50.933]
  Set speed (30.0 mm/s)
  Call Extruder(0.360)
  MoveL 1726 to (490.68, 500.58, 3.4) mm, rotated rx 0 ry 90 rz 0 deg; joints [-12.247, -26.802, 112.007, -16.22, -84.533, 50.566]
  Set speed (120.0 mm/s)
  MoveL 1727 to (490.68, 499.42, 3.4) mm, rotated rx 0 ry 90 rz 0 deg; joints [-12.139, -26.806, 112.036, -16.111, -84.555, 50.55]
  Set speed (30.0 mm/s)
  MoveL 1728 to (499.42, 490.68, 3.4) mm, rotated rx 0 ry 90 rz 0 deg; joints [-11.163, -26.691, 111.215, -15.149, -83.85, 50.657]
  Set speed (120.0 mm/s)
  MoveL 1729 to (500.58, 490.68, 3.4) mm, rotated rx 0 ry 90 rz 0 deg; joints [-11.142, -26.671, 111.077, -15.131, -83.736, 50.686]
  Set speed (30.0 mm/s)
  Call Extruder(0.057)
  MoveL 1730 to (501.97, 492.07, 3.4) mm, rotated rx 0 ry 90 rz 0 deg; joints [-11.244, -26.642, 110.878, -15.239, -83.575, 50.741]
  Set speed (120.0 mm/s)
  MoveL 1731 to (502.07, 492.17, 3.4) mm, rotated rx 0 ry 90 rz 0 deg; joints [-11.252, -26.64, 110.863, -15.247, -83.563, 50.745]
  Set speed (30.0 mm/s)
  Call Extruder(0.262)
  MoveL 1732 to (508.44, 498.54, 3.4) mm, rotated rx 0 ry 90 rz 0 deg; joints [-11.714, -26.5, 109.946, -15.738, -82.827, 51.002]
  MoveL 1733 to (508.56, 498.67, 3.4) mm, rotated rx 0 ry 90 rz 0 deg; joints [-11.723, -26.497, 109.928, -15.747, -82.813, 51.008]
  Set speed (120.0 mm/s)
  MoveL 1734 to (509.32, 490.68, 3.4) mm, rotated rx 0 ry 90 rz 0 deg; joints [-10.985, -26.513, 110.03, -15.001, -82.873, 50.903]
  Set speed (30.0 mm/s)
  Call Extruder(0.767)
  MoveL 1735 to (490.68, 509.32, 3.4) mm, rotated rx 0 ry 90 rz 0 deg; joints [-13.056, -26.77, 111.776, -17.038, -84.362, 50.69]
  MoveL 1736 to (490.56, 509.44, 3.4) mm, rotated rx 0 ry 90 rz 0 deg; joints [-13.07, -26.772, 111.787, -17.052, -84.371, 50.688]
  Set speed (120.0 mm/s)
  MoveL 1737 to (490.4, 509.6, 3.4) mm, rotated rx 0 ry 90 rz 0 deg; joints [-13.088, -26.774, 111.801, -17.069, -84.383, 50.686]
  Set speed (15.0 mm/s)
  Call Extruder(0.559)
  MoveL 1738 to (490.4, 490.4, 3.4) mm, rotated rx 0 ry 90 rz 0 deg; joints [-11.303, -26.839, 112.29, -15.266, -84.748, 50.425]
  MoveL 1739 to (509.6, 490.4, 3.4) mm, rotated rx 0 ry 90 rz 0 deg; joints [-10.955, -26.509, 110.003, -14.971, -82.85, 50.906]
  MoveL 1740 to (509.6, 509.6, 3.4) mm, rotated rx 0 ry 90 rz 0 deg; joints [-12.688, -26.432, 109.519, -16.732, -82.515, 51.214]
  MoveL 1741 to (490.4, 509.6, 3.4) mm, rotated rx 0 ry 90 rz 0 deg; joints [-13.088, -26.774, 111.801, -17.069, -84.383, 50.686]
  Set speed (120.0 mm/s)
  MoveL 1742 to (490.4, 509.2, 3.4) mm, rotated rx 0 ry 90 rz 0 deg; joints [-13.051, -26.775, 111.812, -17.032, -84.391, 50.68]
  Set speed (1000.0 mm/s)
  MoveL 1743 to (490.5, 509.2, 3.4) mm, rotated rx 0 ry 90 rz 0 deg; joints [-13.049, -26.773, 111.8, -17.03, -84.381, 50.683]
  Set speed (1000.0 mm/s)
  MoveL 1744 to (494.72, 492.25, 3.4) mm, rotated rx 0 ry 90 rz 0 deg; joints [-11.395, -26.765, 111.735, -15.37, -84.287, 50.56]
  Set speed (15.0 mm/s)
  Call Extruder(0.034)
  MoveL 1745 to (494.72, 491.09, 3.4) mm, rotated rx 0 ry 90 rz 0 deg; joints [-11.287, -26.768, 111.763, -15.261, -84.308, 50.544]
  Call Extruder(0.075)
  MoveL 1746 to (497.29, 491.09, 3.4) mm, rotated rx 0 ry 90 rz 0 deg; joints [-11.239, -26.726, 111.458, -15.221, -84.054, 50.609]
  Call Extruder(0.034)
  MoveL 1747 to (497.29, 492.25, 3.4) mm, rotated rx 0 ry 90 rz 0 deg; joints [-11.347, -26.722, 111.43, -15.329, -84.033, 50.625]
  Call Extruder(0.075)
  MoveL 1748 to (494.72, 492.25, 3.4) mm, rotated rx 0 ry 90 rz 0 deg; joints [-11.395, -26.765, 111.735, -15.37, -84.287, 50.56]
  Set speed (120.0 mm/s)
  MoveL 1749 to (495.04, 491.94, 3.4) mm, rotated rx 0 ry 90 rz 0 deg; joints [-11.36, -26.76, 111.705, -15.336, -84.261, 50.564]
  Set speed (15.0 mm/s)
  Call Extruder(0.022)
  MoveL 1750 to (495.57, 491.41, 3.4) mm, rotated rx 0 ry 90 rz 0 deg; joints [-11.3, -26.753, 111.654, -15.277, -84.218, 50.57]
  Set speed (120.0 mm/s)
  MoveL 1751 to (496.03, 491.94, 3.4) mm, rotated rx 0 ry 90 rz 0 deg; joints [-11.341, -26.744, 111.587, -15.32, -84.163, 50.589]
  Set speed (15.0 mm/s)
  MoveL 1752 to (496.56, 491.41, 3.4) mm, rotated rx 0 ry 90 rz 0 deg; joints [-11.282, -26.737, 111.537, -15.261, -84.12, 50.595]
  Set speed (120.0 mm/s)
  MoveL 1753 to (501.89, 491.09, 3.4) mm, rotated rx 0 ry 90 rz 0 deg; joints [-11.156, -26.647, 110.911, -15.149, -83.6, 50.725]
  Set speed (15.0 mm/s)
  Call Extruder(0.080)
  MoveL 1754 to (504.63, 491.09, 3.4) mm, rotated rx 0 ry 90 rz 0 deg; joints [-11.106, -26.598, 110.583, -15.108, -83.329, 50.793]
  Call Extruder(0.034)
  MoveL 1755 to (504.63, 492.25, 3.4) mm, rotated rx 0 ry 90 rz 0 deg; joints [-11.212, -26.594, 110.556, -15.216, -83.309, 50.81]
  Call Extruder(0.080)
  MoveL 1756 to (501.89, 492.25, 3.4) mm, rotated rx 0 ry 90 rz 0 deg; joints [-11.262, -26.643, 110.883, -15.258, -83.58, 50.741]
  Call Extruder(0.034)
  MoveL 1757 to (501.89, 491.09, 3.4) mm, rotated rx 0 ry 90 rz 0 deg; joints [-11.156, -26.647, 110.911, -15.149, -83.6, 50.725]
  Set speed (120.0 mm/s)
  MoveL 1758 to (502.5, 491.4, 3.4) mm, rotated rx 0 ry 90 rz 0 deg; joints [-11.173, -26.635, 110.83, -15.169, -83.533, 50.745]
  Set speed (15.0 mm/s)
  Call Extruder(0.012)
  MoveL 1759 to (502.2, 491.71, 3.4) mm, rotated rx 0 ry 90 rz 0 deg; joints [-11.207, -26.639, 110.859, -15.202, -83.558, 50.742]
  Set speed (120.0 mm/s)
  MoveL 1760 to (502.96, 491.94, 3.4) mm, rotated rx 0 ry 90 rz 0 deg; joints [-11.214, -26.625, 110.763, -15.212, -83.479, 50.764]
  Set speed (15.0 mm/s)
  Call Extruder(0.022)
  MoveL 1761 to (503.49, 491.4, 3.4) mm, rotated rx 0 ry 90 rz 0 deg; joints [-11.155, -26.618, 110.712, -15.154, -83.436, 50.77]
  Set speed (120.0 mm/s)
  MoveL 1762 to (503.95, 491.94, 3.4) mm, rotated rx 0 ry 90 rz 0 deg; joints [-11.196, -26.607, 110.644, -15.197, -83.382, 50.789]
  Set speed (15.0 mm/s)
  Call Extruder(0.015)
  MoveL 1763 to (504.31, 491.57, 3.4) mm, rotated rx 0 ry 90 rz 0 deg; joints [-11.156, -26.602, 110.609, -15.158, -83.352, 50.792]
  Set speed (120.0 mm/s)
  MoveL 1764 to (507.69, 498.47, 3.4) mm, rotated rx 0 ry 90 rz 0 deg; joints [-11.721, -26.515, 110.037, -15.742, -82.901, 50.982]
  Set speed (15.0 mm/s)
  Call Extruder(0.035)
  MoveL 1765 to (508.91, 498.46, 3.4) mm, rotated rx 0 ry 90 rz 0 deg; joints [-11.698, -26.492, 109.891, -15.723, -82.782, 51.013]
  Call Extruder(0.070)
  MoveL 1766 to (508.91, 500.87, 3.4) mm, rotated rx 0 ry 90 rz 0 deg; joints [-11.916, -26.482, 109.831, -15.944, -82.74, 51.051]
  Call Extruder(0.035)
  MoveL 1767 to (507.7, 500.87, 3.4) mm, rotated rx 0 ry 90 rz 0 deg; joints [-11.939, -26.505, 109.977, -15.963, -82.859, 51.02]
  Call Extruder(0.070)
  MoveL 1768 to (507.69, 498.47, 3.4) mm, rotated rx 0 ry 90 rz 0 deg; joints [-11.721, -26.515, 110.037, -15.742, -82.901, 50.982]
  Set speed (120.0 mm/s)
  MoveL 1769 to (508.59, 499.17, 3.4) mm, rotated rx 0 ry 90 rz 0 deg; joints [-11.769, -26.495, 109.912, -15.794, -82.801, 51.016]
  Set speed (15.0 mm/s)
  Call Extruder(0.024)
  MoveL 1770 to (508.01, 499.76, 3.4) mm, rotated rx 0 ry 90 rz 0 deg; joints [-11.833, -26.504, 109.967, -15.856, -82.848, 51.011]
  Set speed (120.0 mm/s)
  MoveL 1771 to (508.59, 500.16, 3.4) mm, rotated rx 0 ry 90 rz 0 deg; joints [-11.858, -26.491, 109.887, -15.884, -82.784, 51.032]
  Set speed (15.0 mm/s)
  Call Extruder(0.016)
  MoveL 1772 to (508.2, 500.55, 3.4) mm, rotated rx 0 ry 90 rz 0 deg; joints [-11.901, -26.497, 109.924, -15.926, -82.815, 51.028]
  Set speed (120.0 mm/s)
  MoveL 1773 to (490.68, 490.68, 3.4) mm, rotated rx 0 ry 90 rz 0 deg; joints [-11.324, -26.834, 112.25, -15.288, -84.715, 50.436]
  Set speed (1000.0 mm/s)
  MoveL 1774 to (490.68, 490.68, 3.5) mm, rotated rx 0 ry 90 rz 0 deg; joints [-11.324, -26.845, 112.255, -15.288, -84.71, 50.437]
  Set speed (30.0 mm/s)
  Call Extruder(0.767)
  MoveL 1775 to (509.32, 509.32, 3.5) mm, rotated rx 0 ry 90 rz 0 deg; joints [-12.669, -26.449, 109.566, -16.711, -82.542, 51.203]
  MoveL 1776 to (509.44, 509.44, 3.5) mm, rotated rx 0 ry 90 rz 0 deg; joints [-12.677, -26.446, 109.548, -16.72, -82.528, 51.209]
  Set speed (120.0 mm/s)
  MoveL 1777 to (509.11, 500.79, 3.5) mm, rotated rx 0 ry 90 rz 0 deg; joints [-11.905, -26.489, 109.814, -15.934, -82.717, 51.057]
  Set speed (30.0 mm/s)
  Call Extruder(0.351)
  MoveL 1778 to (500.58, 509.32, 3.5) mm, rotated rx 0 ry 90 rz 0 deg; joints [-12.847, -26.612, 110.61, -16.86, -83.392, 50.966]
  Set speed (120.0 mm/s)
  MoveL 1779 to (499.42, 509.32, 3.5) mm, rotated rx 0 ry 90 rz 0 deg; joints [-12.872, -26.633, 110.748, -16.88, -83.505, 50.934]
  Set speed (30.0 mm/s)
  Call Extruder(0.360)
  MoveL 1780 to (490.68, 500.58, 3.5) mm, rotated rx 0 ry 90 rz 0 deg; joints [-12.247, -26.812, 112.012, -16.22, -84.528, 50.567]
  Set speed (120.0 mm/s)
  MoveL 1781 to (490.68, 499.42, 3.5) mm, rotated rx 0 ry 90 rz 0 deg; joints [-12.139, -26.816, 112.042, -16.111, -84.55, 50.552]
  Set speed (30.0 mm/s)
  MoveL 1782 to (499.42, 490.68, 3.5) mm, rotated rx 0 ry 90 rz 0 deg; joints [-11.163, -26.702, 111.22, -15.149, -83.845, 50.659]
  Set speed (120.0 mm/s)
  MoveL 1783 to (500.58, 490.68, 3.5) mm, rotated rx 0 ry 90 rz 0 deg; joints [-11.142, -26.682, 111.082, -15.131, -83.731, 50.688]
  Set speed (30.0 mm/s)
  Call Extruder(0.055)
  MoveL 1784 to (501.9, 492, 3.5) mm, rotated rx 0 ry 90 rz 0 deg; joints [-11.239, -26.654, 110.893, -15.234, -83.577, 50.74]
  Set speed (120.0 mm/s)
  MoveL 1785 to (502.07, 492.17, 3.5) mm, rotated rx 0 ry 90 rz 0 deg; joints [-11.252, -26.651, 110.869, -15.247, -83.558, 50.746]
  Set speed (30.0 mm/s)
  Call Extruder(0.262)
  MoveL 1786 to (508.44, 498.54, 3.5) mm, rotated rx 0 ry 90 rz 0 deg; joints [-11.714, -26.511, 109.951, -15.738, -82.822, 51.004]
  MoveL 1787 to (508.56, 498.67, 3.5) mm, rotated rx 0 ry 90 rz 0 deg; joints [-11.723, -26.508, 109.933, -15.747, -82.808, 51.009]
  Set speed (120.0 mm/s)
  MoveL 1788 to (509.32, 490.68, 3.5) mm, rotated rx 0 ry 90 rz 0 deg; joints [-10.985, -26.524, 110.035, -15.001, -82.868, 50.904]
  Set speed (30.0 mm/s)
  Call Extruder(0.767)
  MoveL 1789 to (490.68, 509.32, 3.5) mm, rotated rx 0 ry 90 rz 0 deg; joints [-13.056, -26.781, 111.781, -17.038, -84.357, 50.691]
  MoveL 1790 to (490.56, 509.44, 3.5) mm, rotated rx 0 ry 90 rz 0 deg; joints [-13.07, -26.782, 111.792, -17.052, -84.366, 50.69]
  Set speed (120.0 mm/s)
  MoveL 1791 to (490.4, 509.6, 3.5) mm, rotated rx 0 ry 90 rz 0 deg; joints [-13.088, -26.784, 111.806, -17.07, -84.378, 50.688]
  Set speed (15.0 mm/s)
  Call Extruder(0.559)
  MoveL 1792 to (490.4, 490.4, 3.5) mm, rotated rx 0 ry 90 rz 0 deg; joints [-11.303, -26.85, 112.295, -15.266, -84.743, 50.426]
  MoveL 1793 to (509.6, 490.4, 3.5) mm, rotated rx 0 ry 90 rz 0 deg; joints [-10.955, -26.52, 110.008, -14.971, -82.845, 50.907]
  MoveL 1794 to (509.6, 509.6, 3.5) mm, rotated rx 0 ry 90 rz 0 deg; joints [-12.688, -26.443, 109.525, -16.732, -82.51, 51.215]
  MoveL 1795 to (490.4, 509.6, 3.5) mm, rotated rx 0 ry 90 rz 0 deg; joints [-13.088, -26.784, 111.806, -17.07, -84.378, 50.688]
  Set speed (120.0 mm/s)
  MoveL 1796 to (490.4, 509.2, 3.5) mm, rotated rx 0 ry 90 rz 0 deg; joints [-13.051, -26.786, 111.817, -17.032, -84.386, 50.682]
  Set speed (1000.0 mm/s)
  MoveL 1797 to (490.5, 509.2, 3.5) mm, rotated rx 0 ry 90 rz 0 deg; joints [-13.049, -26.784, 111.805, -17.03, -84.376, 50.685]
  Set speed (1000.0 mm/s)
  MoveL 1798 to (494.72, 492.25, 3.5) mm, rotated rx 0 ry 90 rz 0 deg; joints [-11.395, -26.775, 111.741, -15.37, -84.282, 50.561]
  Set speed (15.0 mm/s)
  Call Extruder(0.034)
  MoveL 1799 to (494.72, 491.09, 3.5) mm, rotated rx 0 ry 90 rz 0 deg; joints [-11.287, -26.779, 111.768, -15.261, -84.303, 50.545]
  Call Extruder(0.077)
  MoveL 1800 to (497.35, 491.09, 3.5) mm, rotated rx 0 ry 90 rz 0 deg; joints [-11.238, -26.735, 111.456, -15.22, -84.043, 50.612]
  Call Extruder(0.034)
  MoveL 1801 to (497.35, 492.25, 3.5) mm, rotated rx 0 ry 90 rz 0 deg; joints [-11.346, -26.732, 111.429, -15.329, -84.023, 50.628]
  Call Extruder(0.077)
  MoveL 1802 to (494.72, 492.25, 3.5) mm, rotated rx 0 ry 90 rz 0 deg; joints [-11.395, -26.775, 111.741, -15.37, -84.282, 50.561]
  Set speed (120.0 mm/s)
  MoveL 1803 to (495.37, 491.4, 3.5) mm, rotated rx 0 ry 90 rz 0 deg; joints [-11.304, -26.767, 111.684, -15.281, -84.234, 50.566]
  Set speed (15.0 mm/s)
  Call Extruder(0.022)
  MoveL 1804 to (495.9, 491.94, 3.5) mm, rotated rx 0 ry 90 rz 0 deg; joints [-11.344, -26.757, 111.609, -15.322, -84.172, 50.587]
  Set speed (120.0 mm/s)
  MoveL 1805 to (496.36, 491.41, 3.5) mm, rotated rx 0 ry 90 rz 0 deg; joints [-11.286, -26.751, 111.567, -15.265, -84.136, 50.591]
  Set speed (15.0 mm/s)
  Call Extruder(0.022)
  MoveL 1806 to (496.89, 491.94, 3.5) mm, rotated rx 0 ry 90 rz 0 deg; joints [-11.325, -26.74, 111.491, -15.306, -84.074, 50.612]
  Set speed (120.0 mm/s)
  MoveL 1807 to (501.83, 492.25, 3.5) mm, rotated rx 0 ry 90 rz 0 deg; joints [-11.263, -26.655, 110.896, -15.259, -83.581, 50.741]
  Set speed (15.0 mm/s)
  Call Extruder(0.034)
  MoveL 1808 to (501.83, 491.09, 3.5) mm, rotated rx 0 ry 90 rz 0 deg; joints [-11.157, -26.659, 110.924, -15.151, -83.601, 50.725]
  Call Extruder(0.082)
  MoveL 1809 to (504.63, 491.09, 3.5) mm, rotated rx 0 ry 90 rz 0 deg; joints [-11.106, -26.609, 110.588, -15.108, -83.324, 50.795]
  Call Extruder(0.034)
  MoveL 1810 to (504.63, 492.25, 3.5) mm, rotated rx 0 ry 90 rz 0 deg; joints [-11.212, -26.605, 110.561, -15.216, -83.304, 50.812]
  Call Extruder(0.082)
  MoveL 1811 to (501.83, 492.25, 3.5) mm, rotated rx 0 ry 90 rz 0 deg; joints [-11.263, -26.655, 110.896, -15.259, -83.581, 50.741]
  Set speed (120.0 mm/s)
  MoveL 1812 to (502.29, 491.41, 3.5) mm, rotated rx 0 ry 90 rz 0 deg; joints [-11.177, -26.649, 110.86, -15.173, -83.549, 50.741]
  Set speed (15.0 mm/s)
  Call Extruder(0.022)
  MoveL 1813 to (502.83, 491.94, 3.5) mm, rotated rx 0 ry 90 rz 0 deg; joints [-11.216, -26.638, 110.784, -15.214, -83.488, 50.762]
  Set speed (120.0 mm/s)
  MoveL 1814 to (503.28, 491.41, 3.5) mm, rotated rx 0 ry 90 rz 0 deg; joints [-11.159, -26.632, 110.742, -15.158, -83.451, 50.766]
  Set speed (15.0 mm/s)
  Call Extruder(0.022)
  MoveL 1815 to (503.82, 491.94, 3.5) mm, rotated rx 0 ry 90 rz 0 deg; joints [-11.198, -26.62, 110.666, -15.199, -83.39, 50.787]
  Set speed (120.0 mm/s)
  MoveL 1816 to (507.7, 498.46, 3.5) mm, rotated rx 0 ry 90 rz 0 deg; joints [-11.721, -26.525, 110.043, -15.742, -82.896, 50.983]
  Set speed (15.0 mm/s)
  Call Extruder(0.035)
  MoveL 1817 to (508.91, 498.46, 3.5) mm, rotated rx 0 ry 90 rz 0 deg; joints [-11.698, -26.502, 109.897, -15.723, -82.777, 51.015]
  Call Extruder(0.070)
  MoveL 1818 to (508.91, 500.87, 3.5) mm, rotated rx 0 ry 90 rz 0 deg; joints [-11.916, -26.492, 109.836, -15.944, -82.735, 51.053]
  Call Extruder(0.035)
  MoveL 1819 to (507.69, 500.87, 3.5) mm, rotated rx 0 ry 90 rz 0 deg; joints [-11.939, -26.516, 109.982, -15.963, -82.854, 51.021]
  Call Extruder(0.070)
  MoveL 1820 to (507.7, 498.47, 3.5) mm, rotated rx 0 ry 90 rz 0 deg; joints [-11.721, -26.525, 110.043, -15.742, -82.896, 50.983]
  Call Extruder(0.000)
  MoveL 1821 to (507.7, 498.46, 3.5) mm, rotated rx 0 ry 90 rz 0 deg; joints [-11.721, -26.525, 110.043, -15.742, -82.896, 50.983]
  Set speed (120.0 mm/s)
  MoveL 1822 to (508.01, 499.1, 3.5) mm, rotated rx 0 ry 90 rz 0 deg; joints [-11.773, -26.517, 109.989, -15.796, -82.855, 51.001]
  Set speed (15.0 mm/s)
  Call Extruder(0.024)
  MoveL 1823 to (508.59, 499.68, 3.5) mm, rotated rx 0 ry 90 rz 0 deg; joints [-11.815, -26.503, 109.904, -15.841, -82.787, 51.026]
  Set speed (120.0 mm/s)
  MoveL 1824 to (508.01, 500.09, 3.5) mm, rotated rx 0 ry 90 rz 0 deg; joints [-11.863, -26.513, 109.964, -15.887, -82.837, 51.017]
  Set speed (15.0 mm/s)
  Call Extruder(0.019)
  MoveL 1825 to (508.47, 500.55, 3.5) mm, rotated rx 0 ry 90 rz 0 deg; joints [-11.896, -26.502, 109.897, -15.922, -82.784, 51.037]
  Set speed (120.0 mm/s)
  MoveL 1826 to (490.68, 490.68, 3.5) mm, rotated rx 0 ry 90 rz 0 deg; joints [-11.324, -26.845, 112.255, -15.288, -84.71, 50.437]
  Set speed (1000.0 mm/s)
  MoveL 1827 to (490.68, 490.68, 3.6) mm, rotated rx 0 ry 90 rz 0 deg; joints [-11.324, -26.855, 112.261, -15.288, -84.705, 50.438]
  Set speed (30.0 mm/s)
  Call Extruder(0.767)
  MoveL 1828 to (509.32, 509.32, 3.6) mm, rotated rx 0 ry 90 rz 0 deg; joints [-12.669, -26.46, 109.571, -16.711, -82.537, 51.205]
  MoveL 1829 to (509.44, 509.44, 3.6) mm, rotated rx 0 ry 90 rz 0 deg; joints [-12.677, -26.457, 109.553, -16.721, -82.523, 51.21]
  Set speed (120.0 mm/s)
  MoveL 1830 to (509.11, 500.79, 3.6) mm, rotated rx 0 ry 90 rz 0 deg; joints [-11.905, -26.499, 109.82, -15.934, -82.712, 51.058]
  Set speed (30.0 mm/s)
  Call Extruder(0.351)
  MoveL 1831 to (500.58, 509.32, 3.6) mm, rotated rx 0 ry 90 rz 0 deg; joints [-12.847, -26.623, 110.616, -16.86, -83.387, 50.967]
  Set speed (120.0 mm/s)
  MoveL 1832 to (499.42, 509.32, 3.6) mm, rotated rx 0 ry 90 rz 0 deg; joints [-12.872, -26.643, 110.754, -16.88, -83.5, 50.936]
  Set speed (30.0 mm/s)
  Call Extruder(0.360)
  MoveL 1833 to (490.68, 500.58, 3.6) mm, rotated rx 0 ry 90 rz 0 deg; joints [-12.247, -26.823, 112.017, -16.22, -84.523, 50.569]
  Set speed (120.0 mm/s)
  MoveL 1834 to (490.68, 499.42, 3.6) mm, rotated rx 0 ry 90 rz 0 deg; joints [-12.139, -26.827, 112.047, -16.111, -84.545, 50.553]
  Set speed (30.0 mm/s)
  MoveL 1835 to (499.42, 490.68, 3.6) mm, rotated rx 0 ry 90 rz 0 deg; joints [-11.163, -26.712, 111.225, -15.149, -83.84, 50.66]
  Set speed (120.0 mm/s)
  MoveL 1836 to (500.58, 490.68, 3.6) mm, rotated rx 0 ry 90 rz 0 deg; joints [-11.142, -26.692, 111.087, -15.132, -83.726, 50.689]
  Set speed (30.0 mm/s)
  Call Extruder(0.052)
  MoveL 1837 to (501.84, 491.94, 3.6) mm, rotated rx 0 ry 90 rz 0 deg; joints [-11.235, -26.666, 110.907, -15.23, -83.579, 50.739]
  Set speed (120.0 mm/s)
  MoveL 1838 to (502.07, 492.17, 3.6) mm, rotated rx 0 ry 90 rz 0 deg; joints [-11.252, -26.661, 110.874, -15.248, -83.553, 50.748]
  Set speed (30.0 mm/s)
  Call Extruder(0.262)
  MoveL 1839 to (508.44, 498.54, 3.6) mm, rotated rx 0 ry 90 rz 0 deg; joints [-11.714, -26.521, 109.957, -15.738, -82.817, 51.005]
  MoveL 1840 to (508.56, 498.66, 3.6) mm, rotated rx 0 ry 90 rz 0 deg; joints [-11.723, -26.518, 109.939, -15.747, -82.803, 51.01]
  Set speed (120.0 mm/s)
  MoveL 1841 to (509.32, 490.68, 3.6) mm, rotated rx 0 ry 90 rz 0 deg; joints [-10.985, -26.534, 110.041, -15.001, -82.863, 50.906]
  Set speed (30.0 mm/s)
  Call Extruder(0.767)
  MoveL 1842 to (490.68, 509.32, 3.6) mm, rotated rx 0 ry 90 rz 0 deg; joints [-13.056, -26.791, 111.787, -17.038, -84.352, 50.693]
  MoveL 1843 to (490.56, 509.44, 3.6) mm, rotated rx 0 ry 90 rz 0 deg; joints [-13.07, -26.793, 111.798, -17.052, -84.361, 50.691]
  Set speed (120.0 mm/s)
  MoveL 1844 to (490.4, 509.6, 3.6) mm, rotated rx 0 ry 90 rz 0 deg; joints [-13.088, -26.795, 111.812, -17.07, -84.373, 50.689]
  Set speed (15.0 mm/s)
  Call Extruder(0.559)
  MoveL 1845 to (490.4, 490.4, 3.6) mm, rotated rx 0 ry 90 rz 0 deg; joints [-11.303, -26.861, 112.3, -15.266, -84.738, 50.428]
  MoveL 1846 to (509.6, 490.4, 3.6) mm, rotated rx 0 ry 90 rz 0 deg; joints [-10.955, -26.53, 110.013, -14.972, -82.84, 50.908]
  MoveL 1847 to (509.6, 509.6, 3.6) mm, rotated rx 0 ry 90 rz 0 deg; joints [-12.688, -26.453, 109.53, -16.732, -82.505, 51.217]
  MoveL 1848 to (490.4, 509.6, 3.6) mm, rotated rx 0 ry 90 rz 0 deg; joints [-13.088, -26.795, 111.812, -17.07, -84.373, 50.689]
  Set speed (120.0 mm/s)
  MoveL 1849 to (490.4, 509.2, 3.6) mm, rotated rx 0 ry 90 rz 0 deg; joints [-13.051, -26.796, 111.823, -17.032, -84.381, 50.683]
  Set speed (1000.0 mm/s)
  MoveL 1850 to (490.5, 509.2, 3.6) mm, rotated rx 0 ry 90 rz 0 deg; joints [-13.049, -26.795, 111.811, -17.03, -84.371, 50.686]
  Set speed (1000.0 mm/s)
  MoveL 1851 to (494.72, 492.25, 3.6) mm, rotated rx 0 ry 90 rz 0 deg; joints [-11.395, -26.786, 111.746, -15.371, -84.277, 50.562]
  Set speed (15.0 mm/s)
  Call Extruder(0.034)
  MoveL 1852 to (494.72, 491.09, 3.6) mm, rotated rx 0 ry 90 rz 0 deg; joints [-11.287, -26.79, 111.774, -15.262, -84.298, 50.547]
  Call Extruder(0.078)
  MoveL 1853 to (497.41, 491.09, 3.6) mm, rotated rx 0 ry 90 rz 0 deg; joints [-11.237, -26.745, 111.455, -15.219, -84.032, 50.615]
  Call Extruder(0.034)
  MoveL 1854 to (497.41, 492.25, 3.6) mm, rotated rx 0 ry 90 rz 0 deg; joints [-11.345, -26.741, 111.427, -15.328, -84.012, 50.631]
  Call Extruder(0.078)
  MoveL 1855 to (494.72, 492.25, 3.6) mm, rotated rx 0 ry 90 rz 0 deg; joints [-11.395, -26.786, 111.746, -15.371, -84.277, 50.562]
  Set speed (120.0 mm/s)
  MoveL 1856 to (495.04, 491.94, 3.6) mm, rotated rx 0 ry 90 rz 0 deg; joints [-11.36, -26.782, 111.716, -15.336, -84.251, 50.566]
  Set speed (15.0 mm/s)
  Call Extruder(0.022)
  MoveL 1857 to (495.57, 491.41, 3.6) mm, rotated rx 0 ry 90 rz 0 deg; joints [-11.3, -26.775, 111.665, -15.277, -84.208, 50.573]
  Set speed (120.0 mm/s)
  MoveL 1858 to (496.03, 491.94, 3.6) mm, rotated rx 0 ry 90 rz 0 deg; joints [-11.341, -26.765, 111.598, -15.32, -84.153, 50.592]
  Set speed (15.0 mm/s)
  MoveL 1859 to (496.56, 491.41, 3.6) mm, rotated rx 0 ry 90 rz 0 deg; joints [-11.282, -26.758, 111.548, -15.262, -84.11, 50.598]
  Set speed (120.0 mm/s)
  MoveL 1860 to (501.76, 491.09, 3.6) mm, rotated rx 0 ry 90 rz 0 deg; joints [-11.158, -26.67, 110.936, -15.152, -83.602, 50.725]
  Set speed (15.0 mm/s)
  Call Extruder(0.083)
  MoveL 1861 to (504.63, 491.09, 3.6) mm, rotated rx 0 ry 90 rz 0 deg; joints [-11.106, -26.619, 110.594, -15.108, -83.319, 50.796]
  Call Extruder(0.034)
  MoveL 1862 to (504.63, 492.25, 3.6) mm, rotated rx 0 ry 90 rz 0 deg; joints [-11.212, -26.615, 110.566, -15.216, -83.299, 50.813]
  Call Extruder(0.083)
  MoveL 1863 to (501.77, 492.25, 3.6) mm, rotated rx 0 ry 90 rz 0 deg; joints [-11.265, -26.666, 110.909, -15.26, -83.582, 50.741]
  Call Extruder(0.034)
  MoveL 1864 to (501.76, 491.09, 3.6) mm, rotated rx 0 ry 90 rz 0 deg; joints [-11.158, -26.67, 110.936, -15.152, -83.602, 50.725]
  Set speed (120.0 mm/s)
  MoveL 1865 to (502.5, 491.4, 3.6) mm, rotated rx 0 ry 90 rz 0 deg; joints [-11.173, -26.656, 110.841, -15.17, -83.523, 50.748]
  Set speed (15.0 mm/s)
  Call Extruder(0.018)
  MoveL 1866 to (502.08, 491.83, 3.6) mm, rotated rx 0 ry 90 rz 0 deg; joints [-11.22, -26.662, 110.881, -15.216, -83.558, 50.743]
  Set speed (120.0 mm/s)
  MoveL 1867 to (502.96, 491.94, 3.6) mm, rotated rx 0 ry 90 rz 0 deg; joints [-11.214, -26.646, 110.773, -15.212, -83.469, 50.767]
  Set speed (15.0 mm/s)
  Call Extruder(0.022)
  MoveL 1868 to (503.49, 491.4, 3.6) mm, rotated rx 0 ry 90 rz 0 deg; joints [-11.155, -26.639, 110.722, -15.155, -83.426, 50.772]
  Set speed (120.0 mm/s)
  MoveL 1869 to (503.95, 491.94, 3.6) mm, rotated rx 0 ry 90 rz 0 deg; joints [-11.196, -26.629, 110.655, -15.197, -83.372, 50.791]
  Set speed (15.0 mm/s)
  Call Extruder(0.015)
  MoveL 1870 to (504.31, 491.57, 3.6) mm, rotated rx 0 ry 90 rz 0 deg; joints [-11.156, -26.623, 110.62, -15.158, -83.342, 50.795]
  Set speed (120.0 mm/s)
  MoveL 1871 to (507.7, 498.46, 3.6) mm, rotated rx 0 ry 90 rz 0 deg; joints [-11.721, -26.535, 110.048, -15.742, -82.891, 50.985]
  Set speed (15.0 mm/s)
  Call Extruder(0.035)
  MoveL 1872 to (508.91, 498.46, 3.6) mm, rotated rx 0 ry 90 rz 0 deg; joints [-11.698, -26.513, 109.902, -15.723, -82.772, 51.016]
  Call Extruder(0.070)
  MoveL 1873 to (508.91, 500.87, 3.6) mm, rotated rx 0 ry 90 rz 0 deg; joints [-11.916, -26.503, 109.842, -15.945, -82.73, 51.054]
  Call Extruder(0.035)
  MoveL 1874 to (507.69, 500.87, 3.6) mm, rotated rx 0 ry 90 rz 0 deg; joints [-11.939, -26.526, 109.987, -15.964, -82.849, 51.023]
  Call Extruder(0.070)
  MoveL 1875 to (507.69, 498.46, 3.6) mm, rotated rx 0 ry 90 rz 0 deg; joints [-11.721, -26.535, 110.048, -15.743, -82.891, 50.985]
  Call Extruder(0.000)
  MoveL 1876 to (507.7, 498.46, 3.6) mm, rotated rx 0 ry 90 rz 0 deg; joints [-11.721, -26.535, 110.048, -15.742, -82.891, 50.985]
  Set speed (120.0 mm/s)
  MoveL 1877 to (508.59, 499.17, 3.6) mm, rotated rx 0 ry 90 rz 0 deg; joints [-11.769, -26.516, 109.922, -15.794, -82.791, 51.019]
  Set speed (15.0 mm/s)
  Call Extruder(0.024)
  MoveL 1878 to (508.01, 499.76, 3.6) mm, rotated rx 0 ry 90 rz 0 deg; joints [-11.833, -26.524, 109.978, -15.857, -82.838, 51.013]
  Set speed (120.0 mm/s)
  MoveL 1879 to (508.59, 500.16, 3.6) mm, rotated rx 0 ry 90 rz 0 deg; joints [-11.858, -26.512, 109.897, -15.885, -82.774, 51.035]
  Set speed (15.0 mm/s)
  Call Extruder(0.016)
  MoveL 1880 to (508.2, 500.55, 3.6) mm, rotated rx 0 ry 90 rz 0 deg; joints [-11.901, -26.518, 109.934, -15.927, -82.805, 51.031]
  Set speed (120.0 mm/s)
  MoveL 1881 to (490.68, 490.68, 3.6) mm, rotated rx 0 ry 90 rz 0 deg; joints [-11.324, -26.855, 112.261, -15.288, -84.705, 50.438]
  Set speed (1000.0 mm/s)
  MoveL 1882 to (490.68, 490.68, 3.7) mm, rotated rx 0 ry 90 rz 0 deg; joints [-11.324, -26.866, 112.266, -15.288, -84.7, 50.44]
  Set speed (30.0 mm/s)
  Call Extruder(0.767)
  MoveL 1883 to (509.32, 509.32, 3.7) mm, rotated rx 0 ry 90 rz 0 deg; joints [-12.669, -26.47, 109.577, -16.712, -82.532, 51.206]
  MoveL 1884 to (509.44, 509.44, 3.7) mm, rotated rx 0 ry 90 rz 0 deg; joints [-12.677, -26.467, 109.558, -16.721, -82.518, 51.212]
  Set speed (120.0 mm/s)
  MoveL 1885 to (509.11, 500.79, 3.7) mm, rotated rx 0 ry 90 rz 0 deg; joints [-11.905, -26.51, 109.825, -15.934, -82.707, 51.06]
  Set speed (30.0 mm/s)
  Call Extruder(0.351)
  MoveL 1886 to (500.58, 509.32, 3.7) mm, rotated rx 0 ry 90 rz 0 deg; joints [-12.847, -26.633, 110.621, -16.86, -83.382, 50.969]
  Set speed (120.0 mm/s)
